(* Logix 5000 project; controller reports 1756-L63 rev 20.11; software revision 20.04; part 41 of 52 *)

        [92].log_data[45].valid := 1, [92].log_data[46].time := 3600.0, [92].log_data[46].valid := 1, [92].log_data[47].time := 3600.0, [92].log_data[47].valid := 1, [92].log_data[48].min := 6.688229, [92].log_data[48].max := 6.903953, [92].log_data[48].total := 24394.494, [92].log_data[48].time := 3600.0, [92].log_data[48].maxminute := 57, [92].log_data[48].valid := 1, [92].log_data[49].min := 7.7929306, [92].log_data[49].max := 9.600971, [92].log_data[49].total := 33255.67, [92].log_data[49].time := 3600.0, [92].log_data[49].maxminute := 51, [92].log_data[49].valid := 1, [92].log_data[50].min := 2.0512643, [92].log_data[50].max := 2.1312335, [92].log_data[50].total := 7529.347, [92].log_data[50].time := 3600.0, [92].log_data[50].minminute := 54, [92].log_data[50].valid := 1, [92].log_data[51].time := 3600.0, [92].log_data[51].valid := 1, [92].log_data[52].min := -2.9400024, [92].log_data[52].max := 0.11999512, [92].log_data[52].total := -7606.1123, [92].log_data[52].time := 3600.0, [92].log_data[52].minminute := 5, [92].log_data[52].maxminute := 4, [92].log_data[52].valid := 1, [92].log_data[53].min := -2.5, [92].log_data[53].max := 0.27999878, [92].log_data[53].total := -7261.323, [92].log_data[53].time := 3600.0, [92].log_data[53].minminute := 52, [92].log_data[53].maxminute := 30, [92].log_data[53].valid := 1, [92].log_data[54].max := 0.539, [92].log_data[54].total := 1217.2504, [92].log_data[54].time := 3600.0, [92].log_data[54].minminute := 4, [92].log_data[54].maxminute := 5, [92].log_data[54].valid := 1, [92].log_data[55].max := 0.5365, [92].log_data[55].total := 1254.4075, [92].log_data[55].time := 3600.0, [92].log_data[55].minminute := 8, [92].log_data[55].maxminute := 52, [92].log_data[55].valid := 1, [92].log_data[56].min := 0.15981378, [92].log_data[56].max := 0.16028486, [92].log_data[56].total := 576.022, [92].log_data[56].time := 3600.0, [92].log_data[56].minminute := 1, [92].log_data[56].maxminute := 14, [92].log_data[56].valid := 1, [92].log_data[57].min := 0.23891918, [92].log_data[57].max := 0.23939028,
        [92].log_data[57].total := 860.84656, [92].log_data[57].time := 3600.0, [92].log_data[57].minminute := 12, [92].log_data[57].valid := 1, [92].log_data[58].time := 3600.0, [92].log_data[58].valid := 1, [92].log_data[59].time := 3600.0, [92].log_data[59].valid := 1, [92].log_data[60].valid := 1, [92].log_data[61].valid := 1, [92].log_data[62].valid := 1, [92].log_data[63].valid := 1, [92].log_data[64].valid := 1, [92].log_data[65].valid := 1, [92].log_data[66].valid := 1, [92].log_data[67].valid := 1, [92].log_data[68].valid := 1, [92].log_data[69].valid := 1, [92].log_data[70].valid := 1, [92].log_data[71].valid := 1, [92].log_data[72].valid := 1, [92].log_data[73].valid := 1, [92].log_data[74].valid := 1, [92].log_data[75].valid := 1, [92].log_data[76].valid := 1, [92].log_data[77].valid := 1, [92].log_data[78].valid := 1, [92].log_data[79].valid := 1, [92].log_data[80].valid := 1, [92].log_data[81].valid := 1, [92].log_data[82].valid := 1, [92].log_data[83].valid := 1, [92].log_data[84].valid := 1, [92].log_data[85].valid := 1, [92].log_data[86].valid := 1, [92].log_data[87].valid := 1, [92].log_data[88].valid := 1, [92].log_data[89].valid := 1, [92].log_data[90].valid := 1, [92].log_data[91].valid := 1, [92].log_data[92].valid := 1, [92].log_data[93].valid := 1, [92].log_data[94].valid := 1, [92].log_data[95].valid := 1, [92].log_data[96].valid := 1, [92].log_data[97].valid := 1, [92].log_data[98].valid := 1, [92].log_data[99].valid := 1, [92].log_data[100].valid := 1, [92].log_data[101].valid := 1, [92].log_data[102].valid := 1, [92].log_data[103].valid := 1, [92].log_data[104].valid := 1, [92].log_data[105].valid := 1, [92].log_data[106].valid := 1, [92].log_data[107].valid := 1, [92].log_data[108].valid := 1, [92].log_data[109].valid := 1, [92].log_data[110].valid := 1, [92].log_data[111].valid := 1,
        [92].log_data[112].valid := 1, [92].log_data[113].valid := 1, [92].log_data[114].valid := 1, [92].log_data[115].valid := 1, [92].log_data[116].valid := 1, [92].log_data[117].valid := 1, [92].log_data[118].valid := 1, [92].log_data[119].valid := 1, [92].log_data[120].valid := 1, [92].log_data[121].valid := 1, [92].log_data[122].valid := 1, [92].log_data[123].valid := 1, [92].log_data[124].valid := 1, [92].time.Year := 2023, [92].time.Month := 1, [92].time.Day := 16, [92].time.Hour := 23, [92].time.Minute := 59, [92].time.Second := 59, [93].log_data[0].min := 1.0, [93].log_data[0].max := 1.0, [93].log_data[0].total := 3600.0, [93].log_data[0].time := 3600.0, [93].log_data[0].valid := 1, [93].log_data[1].max := 1.0, [93].log_data[1].total := 72.751, [93].log_data[1].time := 3600.0, [93].log_data[1].minminute := 1, [93].log_data[1].valid := 1, [93].log_data[2].max := 1.0, [93].log_data[2].total := 72.751, [93].log_data[2].time := 3600.0, [93].log_data[2].minminute := 1, [93].log_data[2].valid := 1, [93].log_data[3].time := 3600.0, [93].log_data[3].valid := 1, [93].log_data[4].time := 3600.0, [93].log_data[4].valid := 1, [93].log_data[5].max := 1.0, [93].log_data[5].total := 69.251, [93].log_data[5].time := 3600.0, [93].log_data[5].minminute := 1, [93].log_data[5].valid := 1, [93].log_data[6].time := 3600.0, [93].log_data[6].valid := 1, [93].log_data[7].time := 3600.0, [93].log_data[7].valid := 1, [93].log_data[8].min := 1.0, [93].log_data[8].max := 1.0, [93].log_data[8].total := 3600.0, [93].log_data[8].time := 3600.0, [93].log_data[8].valid := 1, [93].log_data[9].min := 1.0, [93].log_data[9].max := 1.0, [93].log_data[9].total := 3600.0, [93].log_data[9].time := 3600.0, [93].log_data[9].valid := 1, [93].log_data[10].min := 1.0, [93].log_data[10].max := 1.0, [93].log_data[10].total := 3600.0,
        [93].log_data[10].time := 3600.0, [93].log_data[10].valid := 1, [93].log_data[11].time := 3600.0, [93].log_data[11].valid := 1, [93].log_data[12].min := 1.0, [93].log_data[12].max := 1.0, [93].log_data[12].total := 3600.0, [93].log_data[12].time := 3600.0, [93].log_data[12].valid := 1, [93].log_data[13].min := 1.0, [93].log_data[13].max := 1.0, [93].log_data[13].total := 3600.0, [93].log_data[13].time := 3600.0, [93].log_data[13].valid := 1, [93].log_data[14].time := 3600.0, [93].log_data[14].valid := 1, [93].log_data[15].time := 3600.0, [93].log_data[15].valid := 1, [93].log_data[16].time := 3600.0, [93].log_data[16].valid := 1, [93].log_data[17].min := 1.0, [93].log_data[17].max := 1.0, [93].log_data[17].total := 3600.0, [93].log_data[17].time := 3600.0, [93].log_data[17].valid := 1, [93].log_data[18].time := 3600.0, [93].log_data[18].valid := 1, [93].log_data[19].time := 3600.0, [93].log_data[19].valid := 1, [93].log_data[20].time := 3600.0, [93].log_data[20].valid := 1, [93].log_data[21].min := 1.0, [93].log_data[21].max := 1.0, [93].log_data[21].total := 3600.0, [93].log_data[21].time := 3600.0, [93].log_data[21].valid := 1, [93].log_data[22].time := 3600.0, [93].log_data[22].valid := 1, [93].log_data[23].time := 3600.0, [93].log_data[23].valid := 1, [93].log_data[24].time := 3600.0, [93].log_data[24].valid := 1, [93].log_data[25].time := 3600.0, [93].log_data[25].valid := 1, [93].log_data[26].time := 3600.0, [93].log_data[26].valid := 1, [93].log_data[27].time := 3600.0, [93].log_data[27].valid := 1, [93].log_data[28].time := 3600.0, [93].log_data[28].valid := 1, [93].log_data[29].min := 1.0, [93].log_data[29].max := 1.0, [93].log_data[29].total := 3600.0, [93].log_data[29].time := 3600.0, [93].log_data[29].valid := 1, [93].log_data[30].min := 1.0, [93].log_data[30].max := 1.0, [93].log_data[30].total := 3600.0, [93].log_data[30].time := 3600.0, [93].log_data[30].valid := 1,
        [93].log_data[31].max := 1.0, [93].log_data[31].total := 1629.7471, [93].log_data[31].time := 3600.0, [93].log_data[31].maxminute := 8, [93].log_data[31].valid := 1, [93].log_data[32].max := 1.0, [93].log_data[32].total := 1529.249, [93].log_data[32].time := 3600.0, [93].log_data[32].minminute := 7, [93].log_data[32].valid := 1, [93].log_data[33].time := 3600.0, [93].log_data[33].valid := 1, [93].log_data[34].time := 3600.0, [93].log_data[34].valid := 1, [93].log_data[35].max := 1.0, [93].log_data[35].total := 1440.498, [93].log_data[35].time := 3600.0, [93].log_data[35].minminute := 1, [93].log_data[35].valid := 1, [93].log_data[36].max := 1.0, [93].log_data[36].total := 1629.7471, [93].log_data[36].time := 3600.0, [93].log_data[36].maxminute := 2, [93].log_data[36].valid := 1, [93].log_data[37].max := 7.1119633, [93].log_data[37].total := 82.35939, [93].log_data[37].time := 3600.0, [93].log_data[37].valid := 1, [93].log_data[38].time := 3600.0, [93].log_data[38].valid := 1, [93].log_data[39].min := 0.99494183, [93].log_data[39].max := 1.0174367, [93].log_data[39].total := 3603.3508, [93].log_data[39].time := 3600.0, [93].log_data[39].minminute := 5, [93].log_data[39].valid := 1, [93].log_data[40].min := 7.5802555, [93].log_data[40].max := 7.604989, [93].log_data[40].total := 27354.303, [93].log_data[40].time := 3600.0, [93].log_data[40].minminute := 6, [93].log_data[40].maxminute := 8, [93].log_data[40].valid := 1, [93].log_data[41].min := 0.022540038, [93].log_data[41].max := 0.026073486, [93].log_data[41].total := 83.22505, [93].log_data[41].time := 3600.0, [93].log_data[41].minminute := 43, [93].log_data[41].maxminute := 56, [93].log_data[41].valid := 1, [93].log_data[42].min := 2.2917604, [93].log_data[42].max := 2.296236, [93].log_data[42].total := 8259.312, [93].log_data[42].time := 3600.0, [93].log_data[42].minminute := 4, [93].log_data[42].maxminute := 33, [93].log_data[42].valid := 1, [93].log_data[43].min := -0.27999878, [93].log_data[43].max := -0.26000214, [93].log_data[43].total := -1001.4477,
        [93].log_data[43].time := 3600.0, [93].log_data[43].valid := 1, [93].log_data[44].min := -0.3199997, [93].log_data[44].max := -0.30000305, [93].log_data[44].total := -1080.1111, [93].log_data[44].time := 3600.0, [93].log_data[44].minminute := 37, [93].log_data[44].valid := 1, [93].log_data[45].time := 3600.0, [93].log_data[45].valid := 1, [93].log_data[46].time := 3600.0, [93].log_data[46].valid := 1, [93].log_data[47].time := 3600.0, [93].log_data[47].valid := 1, [93].log_data[48].min := 6.587924, [93].log_data[48].max := 6.9380293, [93].log_data[48].total := 24235.338, [93].log_data[48].time := 3600.0, [93].log_data[48].minminute := 26, [93].log_data[48].maxminute := 1, [93].log_data[48].valid := 1, [93].log_data[49].min := 6.965759, [93].log_data[49].max := 9.442367, [93].log_data[49].total := 29303.482, [93].log_data[49].time := 3600.0, [93].log_data[49].minminute := 22, [93].log_data[49].maxminute := 59, [93].log_data[49].valid := 1, [93].log_data[50].min := 2.0797658, [93].log_data[50].max := 2.1550238, [93].log_data[50].total := 7630.34, [93].log_data[50].time := 3600.0, [93].log_data[50].minminute := 59, [93].log_data[50].maxminute := 3, [93].log_data[50].valid := 1, [93].log_data[51].time := 3600.0, [93].log_data[51].valid := 1, [93].log_data[52].min := -3.1200027, [93].log_data[52].max := 0.11999512, [93].log_data[52].total := -7898.7217, [93].log_data[52].time := 3600.0, [93].log_data[52].minminute := 29, [93].log_data[52].maxminute := 7, [93].log_data[52].valid := 1, [93].log_data[53].min := -2.5200043, [93].log_data[53].max := 0.27999878, [93].log_data[53].total := -7128.1104, [93].log_data[53].time := 3600.0, [93].log_data[53].minminute := 13, [93].log_data[53].maxminute := 23, [93].log_data[53].valid := 1, [93].log_data[54].max := 0.5565, [93].log_data[54].total := 1254.5945, [93].log_data[54].time := 3600.0, [93].log_data[54].minminute := 7, [93].log_data[54].maxminute := 30, [93].log_data[54].valid := 1, [93].log_data[55].max := 0.519, [93].log_data[55].total := 1216.6926, [93].log_data[55].time := 3600.0,
        [93].log_data[55].minminute := 1, [93].log_data[55].maxminute := 44, [93].log_data[55].valid := 1, [93].log_data[56].min := 0.15981378, [93].log_data[56].max := 0.16024561, [93].log_data[56].total := 575.9473, [93].log_data[56].time := 3600.0, [93].log_data[56].minminute := 24, [93].log_data[56].maxminute := 41, [93].log_data[56].valid := 1, [93].log_data[57].min := 0.23754516, [93].log_data[57].max := 0.23935102, [93].log_data[57].total := 858.23517, [93].log_data[57].time := 3600.0, [93].log_data[57].minminute := 39, [93].log_data[57].maxminute := 21, [93].log_data[57].valid := 1, [93].log_data[58].time := 3600.0, [93].log_data[58].valid := 1, [93].log_data[59].time := 3600.0, [93].log_data[59].valid := 1, [93].log_data[60].valid := 1, [93].log_data[61].valid := 1, [93].log_data[62].valid := 1, [93].log_data[63].valid := 1, [93].log_data[64].valid := 1, [93].log_data[65].valid := 1, [93].log_data[66].valid := 1, [93].log_data[67].valid := 1, [93].log_data[68].valid := 1, [93].log_data[69].valid := 1, [93].log_data[70].valid := 1, [93].log_data[71].valid := 1, [93].log_data[72].valid := 1, [93].log_data[73].valid := 1, [93].log_data[74].valid := 1, [93].log_data[75].valid := 1, [93].log_data[76].valid := 1, [93].log_data[77].valid := 1, [93].log_data[78].valid := 1, [93].log_data[79].valid := 1, [93].log_data[80].valid := 1, [93].log_data[81].valid := 1, [93].log_data[82].valid := 1, [93].log_data[83].valid := 1, [93].log_data[84].valid := 1, [93].log_data[85].valid := 1, [93].log_data[86].valid := 1, [93].log_data[87].valid := 1, [93].log_data[88].valid := 1, [93].log_data[89].valid := 1, [93].log_data[90].valid := 1, [93].log_data[91].valid := 1, [93].log_data[92].valid := 1, [93].log_data[93].valid := 1, [93].log_data[94].valid := 1, [93].log_data[95].valid := 1, [93].log_data[96].valid := 1, [93].log_data[97].valid := 1, [93].log_data[98].valid := 1,
        [93].log_data[99].valid := 1, [93].log_data[100].valid := 1, [93].log_data[101].valid := 1, [93].log_data[102].valid := 1, [93].log_data[103].valid := 1, [93].log_data[104].valid := 1, [93].log_data[105].valid := 1, [93].log_data[106].valid := 1, [93].log_data[107].valid := 1, [93].log_data[108].valid := 1, [93].log_data[109].valid := 1, [93].log_data[110].valid := 1, [93].log_data[111].valid := 1, [93].log_data[112].valid := 1, [93].log_data[113].valid := 1, [93].log_data[114].valid := 1, [93].log_data[115].valid := 1, [93].log_data[116].valid := 1, [93].log_data[117].valid := 1, [93].log_data[118].valid := 1, [93].log_data[119].valid := 1, [93].log_data[120].valid := 1, [93].log_data[121].valid := 1, [93].log_data[122].valid := 1, [93].log_data[123].valid := 1, [93].log_data[124].valid := 1, [93].time.Year := 2023, [93].time.Month := 1, [93].time.Day := 17, [93].time.Minute := 59, [93].time.Second := 59, [94].log_data[0].min := 1.0, [94].log_data[0].max := 1.0, [94].log_data[0].total := 3600.0, [94].log_data[0].time := 3600.0, [94].log_data[0].valid := 1, [94].log_data[1].time := 3600.0, [94].log_data[1].valid := 1, [94].log_data[2].time := 3600.0, [94].log_data[2].valid := 1, [94].log_data[3].time := 3600.0, [94].log_data[3].valid := 1, [94].log_data[4].time := 3600.0, [94].log_data[4].valid := 1, [94].log_data[5].time := 3600.0, [94].log_data[5].valid := 1, [94].log_data[6].time := 3600.0, [94].log_data[6].valid := 1, [94].log_data[7].time := 3600.0, [94].log_data[7].valid := 1, [94].log_data[8].max := 1.0, [94].log_data[8].total := 2725.751, [94].log_data[8].time := 3600.0, [94].log_data[8].minminute := 45, [94].log_data[8].valid := 1, [94].log_data[9].max := 1.0, [94].log_data[9].total := 2725.751, [94].log_data[9].time := 3600.0, [94].log_data[9].minminute := 45, [94].log_data[9].valid := 1,
        [94].log_data[10].min := 1.0, [94].log_data[10].max := 1.0, [94].log_data[10].total := 3600.0, [94].log_data[10].time := 3600.0, [94].log_data[10].valid := 1, [94].log_data[11].time := 3600.0, [94].log_data[11].valid := 1, [94].log_data[12].min := 1.0, [94].log_data[12].max := 1.0, [94].log_data[12].total := 3600.0, [94].log_data[12].time := 3600.0, [94].log_data[12].valid := 1, [94].log_data[13].min := 1.0, [94].log_data[13].max := 1.0, [94].log_data[13].total := 3600.0, [94].log_data[13].time := 3600.0, [94].log_data[13].valid := 1, [94].log_data[14].time := 3600.0, [94].log_data[14].valid := 1, [94].log_data[15].time := 3600.0, [94].log_data[15].valid := 1, [94].log_data[16].time := 3600.0, [94].log_data[16].valid := 1, [94].log_data[17].min := 1.0, [94].log_data[17].max := 1.0, [94].log_data[17].total := 3600.0, [94].log_data[17].time := 3600.0, [94].log_data[17].valid := 1, [94].log_data[18].time := 3600.0, [94].log_data[18].valid := 1, [94].log_data[19].time := 3600.0, [94].log_data[19].valid := 1, [94].log_data[20].time := 3600.0, [94].log_data[20].valid := 1, [94].log_data[21].min := 1.0, [94].log_data[21].max := 1.0, [94].log_data[21].total := 3600.0, [94].log_data[21].time := 3600.0, [94].log_data[21].valid := 1, [94].log_data[22].time := 3600.0, [94].log_data[22].valid := 1, [94].log_data[23].time := 3600.0, [94].log_data[23].valid := 1, [94].log_data[24].time := 3600.0, [94].log_data[24].valid := 1, [94].log_data[25].time := 3600.0, [94].log_data[25].valid := 1, [94].log_data[26].time := 3600.0, [94].log_data[26].valid := 1, [94].log_data[27].time := 3600.0, [94].log_data[27].valid := 1, [94].log_data[28].time := 3600.0, [94].log_data[28].valid := 1, [94].log_data[29].min := 1.0, [94].log_data[29].max := 1.0, [94].log_data[29].total := 3600.0, [94].log_data[29].time := 3600.0, [94].log_data[29].valid := 1, [94].log_data[30].min := 1.0, [94].log_data[30].max := 1.0,
        [94].log_data[30].total := 3600.0, [94].log_data[30].time := 3600.0, [94].log_data[30].valid := 1, [94].log_data[31].max := 1.0, [94].log_data[31].total := 1086.498, [94].log_data[31].time := 3600.0, [94].log_data[31].maxminute := 11, [94].log_data[31].valid := 1, [94].log_data[32].max := 1.0, [94].log_data[32].total := 1201.7471, [94].log_data[32].time := 3600.0, [94].log_data[32].maxminute := 1, [94].log_data[32].valid := 1, [94].log_data[33].time := 3600.0, [94].log_data[33].valid := 1, [94].log_data[34].time := 3600.0, [94].log_data[34].valid := 1, [94].log_data[35].max := 1.0, [94].log_data[35].total := 1289.998, [94].log_data[35].time := 3600.0, [94].log_data[35].minminute := 4, [94].log_data[35].valid := 1, [94].log_data[36].max := 1.0, [94].log_data[36].total := 1086.498, [94].log_data[36].time := 3600.0, [94].log_data[36].maxminute := 5, [94].log_data[36].valid := 1, [94].log_data[37].time := 3600.0, [94].log_data[37].valid := 1, [94].log_data[38].time := 3600.0, [94].log_data[38].valid := 1, [94].log_data[39].min := 0.9944707, [94].log_data[39].max := 1.0054238, [94].log_data[39].total := 3603.0454, [94].log_data[39].time := 3600.0, [94].log_data[39].minminute := 12, [94].log_data[39].valid := 1, [94].log_data[40].min := 7.591522, [94].log_data[40].max := 7.604989, [94].log_data[40].total := 27355.736, [94].log_data[40].time := 3600.0, [94].log_data[40].minminute := 48, [94].log_data[40].maxminute := 54, [94].log_data[40].valid := 1, [94].log_data[41].min := 0.02273633, [94].log_data[41].max := 0.026073486, [94].log_data[41].total := 83.72127, [94].log_data[41].time := 3600.0, [94].log_data[41].minminute := 9, [94].log_data[41].valid := 1, [94].log_data[42].min := 2.2911716, [94].log_data[42].max := 2.2963536, [94].log_data[42].total := 8259.223, [94].log_data[42].time := 3600.0, [94].log_data[42].minminute := 33, [94].log_data[42].maxminute := 35, [94].log_data[42].valid := 1, [94].log_data[43].min := -0.27999878, [94].log_data[43].max := -0.26000214, [94].log_data[43].total := -1002.2216,
        [94].log_data[43].time := 3600.0, [94].log_data[43].valid := 1, [94].log_data[44].min := -0.3199997, [94].log_data[44].max := -0.30000305, [94].log_data[44].total := -1080.0962, [94].log_data[44].time := 3600.0, [94].log_data[44].minminute := 20, [94].log_data[44].valid := 1, [94].log_data[45].time := 3600.0, [94].log_data[45].valid := 1, [94].log_data[46].time := 3600.0, [94].log_data[46].valid := 1, [94].log_data[47].time := 3600.0, [94].log_data[47].valid := 1, [94].log_data[48].min := 6.7649, [94].log_data[48].max := 6.7800145, [94].log_data[48].total := 24376.885, [94].log_data[48].time := 3600.0, [94].log_data[48].minminute := 50, [94].log_data[48].maxminute := 1, [94].log_data[48].valid := 1, [94].log_data[49].min := 9.429412, [94].log_data[49].max := 9.602148, [94].log_data[49].total := 34382.223, [94].log_data[49].time := 3600.0, [94].log_data[49].maxminute := 32, [94].log_data[49].valid := 1, [94].log_data[50].min := 1.9999144, [94].log_data[50].max := 2.1160402, [94].log_data[50].total := 7404.776, [94].log_data[50].time := 3600.0, [94].log_data[50].minminute := 45, [94].log_data[50].maxminute := 59, [94].log_data[50].valid := 1, [94].log_data[51].time := 3600.0, [94].log_data[51].valid := 1, [94].log_data[52].min := -2.9400024, [94].log_data[52].max := 0.11999512, [94].log_data[52].total := -6819.65, [94].log_data[52].time := 3600.0, [94].log_data[52].minminute := 12, [94].log_data[52].valid := 1, [94].log_data[53].min := -2.4800034, [94].log_data[53].max := 0.27999878, [94].log_data[53].total := -6552.212, [94].log_data[53].time := 3600.0, [94].log_data[53].minminute := 2, [94].log_data[53].maxminute := 5, [94].log_data[53].valid := 1, [94].log_data[54].max := 0.524, [94].log_data[54].total := 906.4553, [94].log_data[54].time := 3600.0, [94].log_data[54].maxminute := 12, [94].log_data[54].valid := 1, [94].log_data[55].max := 0.517, [94].log_data[55].total := 943.5342, [94].log_data[55].time := 3600.0, [94].log_data[55].minminute := 4, [94].log_data[55].maxminute := 5, [94].log_data[55].valid := 1,
        [94].log_data[56].min := 0.15985303, [94].log_data[56].max := 0.16024561, [94].log_data[56].total := 575.978, [94].log_data[56].time := 3600.0, [94].log_data[56].minminute := 5, [94].log_data[56].maxminute := 25, [94].log_data[56].valid := 1, [94].log_data[57].min := 0.23754516, [94].log_data[57].max := 0.237977, [94].log_data[57].total := 855.8624, [94].log_data[57].time := 3600.0, [94].log_data[57].minminute := 21, [94].log_data[57].maxminute := 44, [94].log_data[57].valid := 1, [94].log_data[58].time := 3600.0, [94].log_data[58].valid := 1, [94].log_data[59].time := 3600.0, [94].log_data[59].valid := 1, [94].log_data[60].valid := 1, [94].log_data[61].valid := 1, [94].log_data[62].valid := 1, [94].log_data[63].valid := 1, [94].log_data[64].valid := 1, [94].log_data[65].valid := 1, [94].log_data[66].valid := 1, [94].log_data[67].valid := 1, [94].log_data[68].valid := 1, [94].log_data[69].valid := 1, [94].log_data[70].valid := 1, [94].log_data[71].valid := 1, [94].log_data[72].valid := 1, [94].log_data[73].valid := 1, [94].log_data[74].valid := 1, [94].log_data[75].valid := 1, [94].log_data[76].valid := 1, [94].log_data[77].valid := 1, [94].log_data[78].valid := 1, [94].log_data[79].valid := 1, [94].log_data[80].valid := 1, [94].log_data[81].valid := 1, [94].log_data[82].valid := 1, [94].log_data[83].valid := 1, [94].log_data[84].valid := 1, [94].log_data[85].valid := 1, [94].log_data[86].valid := 1, [94].log_data[87].valid := 1, [94].log_data[88].valid := 1, [94].log_data[89].valid := 1, [94].log_data[90].valid := 1, [94].log_data[91].valid := 1, [94].log_data[92].valid := 1, [94].log_data[93].valid := 1, [94].log_data[94].valid := 1, [94].log_data[95].valid := 1, [94].log_data[96].valid := 1, [94].log_data[97].valid := 1, [94].log_data[98].valid := 1, [94].log_data[99].valid := 1, [94].log_data[100].valid := 1, [94].log_data[101].valid := 1,
        [94].log_data[102].valid := 1, [94].log_data[103].valid := 1, [94].log_data[104].valid := 1, [94].log_data[105].valid := 1, [94].log_data[106].valid := 1, [94].log_data[107].valid := 1, [94].log_data[108].valid := 1, [94].log_data[109].valid := 1, [94].log_data[110].valid := 1, [94].log_data[111].valid := 1, [94].log_data[112].valid := 1, [94].log_data[113].valid := 1, [94].log_data[114].valid := 1, [94].log_data[115].valid := 1, [94].log_data[116].valid := 1, [94].log_data[117].valid := 1, [94].log_data[118].valid := 1, [94].log_data[119].valid := 1, [94].log_data[120].valid := 1, [94].log_data[121].valid := 1, [94].log_data[122].valid := 1, [94].log_data[123].valid := 1, [94].log_data[124].valid := 1, [94].time.Year := 2023, [94].time.Month := 1, [94].time.Day := 17, [94].time.Hour := 1, [94].time.Minute := 59, [94].time.Second := 59, [95].log_data[0].min := 1.0, [95].log_data[0].max := 1.0, [95].log_data[0].total := 3600.0, [95].log_data[0].time := 3600.0, [95].log_data[0].valid := 1, [95].log_data[1].max := 1.0, [95].log_data[1].total := 526.5, [95].log_data[1].time := 3600.0, [95].log_data[1].maxminute := 3, [95].log_data[1].valid := 1, [95].log_data[2].max := 1.0, [95].log_data[2].total := 523.0, [95].log_data[2].time := 3600.0, [95].log_data[2].maxminute := 3, [95].log_data[2].valid := 1, [95].log_data[3].time := 3600.0, [95].log_data[3].valid := 1, [95].log_data[4].time := 3600.0, [95].log_data[4].valid := 1, [95].log_data[5].max := 1.0, [95].log_data[5].total := 233.0, [95].log_data[5].time := 3600.0, [95].log_data[5].maxminute := 5, [95].log_data[5].valid := 1, [95].log_data[6].time := 3600.0, [95].log_data[6].valid := 1, [95].log_data[7].time := 3600.0, [95].log_data[7].valid := 1, [95].log_data[8].max := 1.0, [95].log_data[8].total := 3184.749, [95].log_data[8].time := 3600.0,
        [95].log_data[8].maxminute := 6, [95].log_data[8].valid := 1, [95].log_data[9].max := 1.0, [95].log_data[9].total := 3181.249, [95].log_data[9].time := 3600.0, [95].log_data[9].maxminute := 6, [95].log_data[9].valid := 1, [95].log_data[10].min := 1.0, [95].log_data[10].max := 1.0, [95].log_data[10].total := 3600.0, [95].log_data[10].time := 3600.0, [95].log_data[10].valid := 1, [95].log_data[11].time := 3600.0, [95].log_data[11].valid := 1, [95].log_data[12].min := 1.0, [95].log_data[12].max := 1.0, [95].log_data[12].total := 3600.0, [95].log_data[12].time := 3600.0, [95].log_data[12].valid := 1, [95].log_data[13].min := 1.0, [95].log_data[13].max := 1.0, [95].log_data[13].total := 3600.0, [95].log_data[13].time := 3600.0, [95].log_data[13].valid := 1, [95].log_data[14].time := 3600.0, [95].log_data[14].valid := 1, [95].log_data[15].time := 3600.0, [95].log_data[15].valid := 1, [95].log_data[16].time := 3600.0, [95].log_data[16].valid := 1, [95].log_data[17].min := 1.0, [95].log_data[17].max := 1.0, [95].log_data[17].total := 3600.0, [95].log_data[17].time := 3600.0, [95].log_data[17].valid := 1, [95].log_data[18].time := 3600.0, [95].log_data[18].valid := 1, [95].log_data[19].time := 3600.0, [95].log_data[19].valid := 1, [95].log_data[20].time := 3600.0, [95].log_data[20].valid := 1, [95].log_data[21].min := 1.0, [95].log_data[21].max := 1.0, [95].log_data[21].total := 3600.0, [95].log_data[21].time := 3600.0, [95].log_data[21].valid := 1, [95].log_data[22].time := 3600.0, [95].log_data[22].valid := 1, [95].log_data[23].time := 3600.0, [95].log_data[23].valid := 1, [95].log_data[24].time := 3600.0, [95].log_data[24].valid := 1, [95].log_data[25].time := 3600.0, [95].log_data[25].valid := 1, [95].log_data[26].time := 3600.0, [95].log_data[26].valid := 1, [95].log_data[27].time := 3600.0, [95].log_data[27].valid := 1, [95].log_data[28].time := 3600.0, [95].log_data[28].valid := 1,
        [95].log_data[29].min := 1.0, [95].log_data[29].max := 1.0, [95].log_data[29].total := 3600.0, [95].log_data[29].time := 3600.0, [95].log_data[29].valid := 1, [95].log_data[30].min := 1.0, [95].log_data[30].max := 1.0, [95].log_data[30].total := 3600.0, [95].log_data[30].time := 3600.0, [95].log_data[30].valid := 1, [95].log_data[31].max := 1.0, [95].log_data[31].total := 1514.247, [95].log_data[31].time := 3600.0, [95].log_data[31].maxminute := 7, [95].log_data[31].valid := 1, [95].log_data[32].max := 1.0, [95].log_data[32].total := 1221.998, [95].log_data[32].time := 3600.0, [95].log_data[32].maxminute := 15, [95].log_data[32].valid := 1, [95].log_data[33].time := 3600.0, [95].log_data[33].valid := 1, [95].log_data[34].time := 3600.0, [95].log_data[34].valid := 1, [95].log_data[35].max := 1.0, [95].log_data[35].total := 1593.7471, [95].log_data[35].time := 3600.0, [95].log_data[35].maxminute := 9, [95].log_data[35].valid := 1, [95].log_data[36].max := 1.0, [95].log_data[36].total := 1139.247, [95].log_data[36].time := 3600.0, [95].log_data[36].maxminute := 7, [95].log_data[36].valid := 1, [95].log_data[37].max := 7.4978714, [95].log_data[37].total := 3407.6616, [95].log_data[37].time := 3600.0, [95].log_data[37].maxminute := 4, [95].log_data[37].valid := 1, [95].log_data[38].time := 3600.0, [95].log_data[38].valid := 1, [95].log_data[39].min := 0.99282193, [95].log_data[39].max := 1.0216767, [95].log_data[39].total := 3605.1196, [95].log_data[39].time := 3600.0, [95].log_data[39].minminute := 54, [95].log_data[39].maxminute := 10, [95].log_data[39].valid := 1, [95].log_data[40].min := 7.591522, [95].log_data[40].max := 7.605263, [95].log_data[40].total := 27359.295, [95].log_data[40].time := 3600.0, [95].log_data[40].minminute := 6, [95].log_data[40].maxminute := 11, [95].log_data[40].valid := 1, [95].log_data[41].min := 0.022540038, [95].log_data[41].max := 0.027054932, [95].log_data[41].total := 83.72717, [95].log_data[41].time := 3600.0, [95].log_data[41].minminute := 19,
        [95].log_data[41].maxminute := 36, [95].log_data[41].valid := 1, [95].log_data[42].min := 2.291525, [95].log_data[42].max := 2.296118, [95].log_data[42].total := 8259.106, [95].log_data[42].time := 3600.0, [95].log_data[42].minminute := 11, [95].log_data[42].maxminute := 11, [95].log_data[42].valid := 1, [95].log_data[43].min := -0.27999878, [95].log_data[43].max := -0.26000214, [95].log_data[43].total := -976.2031, [95].log_data[43].time := 3600.0, [95].log_data[43].valid := 1, [95].log_data[44].min := -0.30000305, [95].log_data[44].max := -0.30000305, [95].log_data[44].total := -1080.0911, [95].log_data[44].time := 3600.0, [95].log_data[44].valid := 1, [95].log_data[45].time := 3600.0, [95].log_data[45].valid := 1, [95].log_data[46].time := 3600.0, [95].log_data[46].valid := 1, [95].log_data[47].time := 3600.0, [95].log_data[47].valid := 1, [95].log_data[48].min := 6.589573, [95].log_data[48].max := 6.9465485, [95].log_data[48].total := 24249.084, [95].log_data[48].time := 3600.0, [95].log_data[48].minminute := 37, [95].log_data[48].maxminute := 12, [95].log_data[48].valid := 1, [95].log_data[49].min := 6.8835125, [95].log_data[49].max := 9.557198, [95].log_data[49].total := 29212.176, [95].log_data[49].time := 3600.0, [95].log_data[49].minminute := 32, [95].log_data[49].maxminute := 2, [95].log_data[49].valid := 1, [95].log_data[50].min := 2.0484376, [95].log_data[50].max := 2.150313, [95].log_data[50].total := 7525.7383, [95].log_data[50].time := 3600.0, [95].log_data[50].minminute := 59, [95].log_data[50].maxminute := 6, [95].log_data[50].valid := 1, [95].log_data[51].time := 3600.0, [95].log_data[51].valid := 1, [95].log_data[52].min := -4.3399963, [95].log_data[52].max := 0.11999512, [95].log_data[52].total := -7494.401, [95].log_data[52].time := 3600.0, [95].log_data[52].minminute := 7, [95].log_data[52].maxminute := 14, [95].log_data[52].valid := 1, [95].log_data[53].min := -3.9399948, [95].log_data[53].max := 0.27999878, [95].log_data[53].total := -6960.026, [95].log_data[53].time := 3600.0, [95].log_data[53].minminute := 7,
        [95].log_data[53].maxminute := 19, [95].log_data[53].valid := 1, [95].log_data[54].max := 0.5355, [95].log_data[54].total := 1083.5779, [95].log_data[54].time := 3600.0, [95].log_data[54].maxminute := 26, [95].log_data[54].valid := 1, [95].log_data[55].max := 0.518, [95].log_data[55].total := 1081.9321, [95].log_data[55].time := 3600.0, [95].log_data[55].maxminute := 30, [95].log_data[55].valid := 1, [95].log_data[56].min := 0.15973525, [95].log_data[56].max := 0.16020635, [95].log_data[56].total := 575.83905, [95].log_data[56].time := 3600.0, [95].log_data[56].minminute := 37, [95].log_data[56].maxminute := 4, [95].log_data[56].valid := 1, [95].log_data[57].min := 0.2362104, [95].log_data[57].max := 0.23801626, [95].log_data[57].total := 854.2079, [95].log_data[57].time := 3600.0, [95].log_data[57].minminute := 52, [95].log_data[57].maxminute := 15, [95].log_data[57].valid := 1, [95].log_data[58].time := 3600.0, [95].log_data[58].valid := 1, [95].log_data[59].time := 3600.0, [95].log_data[59].valid := 1, [95].log_data[60].valid := 1, [95].log_data[61].valid := 1, [95].log_data[62].valid := 1, [95].log_data[63].valid := 1, [95].log_data[64].valid := 1, [95].log_data[65].valid := 1, [95].log_data[66].valid := 1, [95].log_data[67].valid := 1, [95].log_data[68].valid := 1, [95].log_data[69].valid := 1, [95].log_data[70].valid := 1, [95].log_data[71].valid := 1, [95].log_data[72].valid := 1, [95].log_data[73].valid := 1, [95].log_data[74].valid := 1, [95].log_data[75].valid := 1, [95].log_data[76].valid := 1, [95].log_data[77].valid := 1, [95].log_data[78].valid := 1, [95].log_data[79].valid := 1, [95].log_data[80].valid := 1, [95].log_data[81].valid := 1, [95].log_data[82].valid := 1, [95].log_data[83].valid := 1, [95].log_data[84].valid := 1, [95].log_data[85].valid := 1, [95].log_data[86].valid := 1, [95].log_data[87].valid := 1, [95].log_data[88].valid := 1, [95].log_data[89].valid := 1,
        [95].log_data[90].valid := 1, [95].log_data[91].valid := 1, [95].log_data[92].valid := 1, [95].log_data[93].valid := 1, [95].log_data[94].valid := 1, [95].log_data[95].valid := 1, [95].log_data[96].valid := 1, [95].log_data[97].valid := 1, [95].log_data[98].valid := 1, [95].log_data[99].valid := 1, [95].log_data[100].valid := 1, [95].log_data[101].valid := 1, [95].log_data[102].valid := 1, [95].log_data[103].valid := 1, [95].log_data[104].valid := 1, [95].log_data[105].valid := 1, [95].log_data[106].valid := 1, [95].log_data[107].valid := 1, [95].log_data[108].valid := 1, [95].log_data[109].valid := 1, [95].log_data[110].valid := 1, [95].log_data[111].valid := 1, [95].log_data[112].valid := 1, [95].log_data[113].valid := 1, [95].log_data[114].valid := 1, [95].log_data[115].valid := 1, [95].log_data[116].valid := 1, [95].log_data[117].valid := 1, [95].log_data[118].valid := 1, [95].log_data[119].valid := 1, [95].log_data[120].valid := 1, [95].log_data[121].valid := 1, [95].log_data[122].valid := 1, [95].log_data[123].valid := 1, [95].log_data[124].valid := 1, [95].time.Year := 2023, [95].time.Month := 1, [95].time.Day := 17, [95].time.Hour := 2, [95].time.Minute := 59, [95].time.Second := 59, [96].log_data[0].min := 1.0, [96].log_data[0].max := 1.0, [96].log_data[0].total := 3600.0, [96].log_data[0].time := 3600.0, [96].log_data[0].valid := 1, [96].log_data[1].time := 3600.0, [96].log_data[1].valid := 1, [96].log_data[2].time := 3600.0, [96].log_data[2].valid := 1, [96].log_data[3].time := 3600.0, [96].log_data[3].valid := 1, [96].log_data[4].time := 3600.0, [96].log_data[4].valid := 1, [96].log_data[5].time := 3600.0, [96].log_data[5].valid := 1, [96].log_data[6].time := 3600.0, [96].log_data[6].valid := 1, [96].log_data[7].time := 3600.0, [96].log_data[7].valid := 1,
        [96].log_data[8].max := 1.0, [96].log_data[8].total := 2187.751, [96].log_data[8].time := 3600.0, [96].log_data[8].minminute := 36, [96].log_data[8].valid := 1, [96].log_data[9].max := 1.0, [96].log_data[9].total := 2187.751, [96].log_data[9].time := 3600.0, [96].log_data[9].minminute := 36, [96].log_data[9].valid := 1, [96].log_data[10].min := 1.0, [96].log_data[10].max := 1.0, [96].log_data[10].total := 3600.0, [96].log_data[10].time := 3600.0, [96].log_data[10].valid := 1, [96].log_data[11].time := 3600.0, [96].log_data[11].valid := 1, [96].log_data[12].min := 1.0, [96].log_data[12].max := 1.0, [96].log_data[12].total := 3600.0, [96].log_data[12].time := 3600.0, [96].log_data[12].valid := 1, [96].log_data[13].min := 1.0, [96].log_data[13].max := 1.0, [96].log_data[13].total := 3600.0, [96].log_data[13].time := 3600.0, [96].log_data[13].valid := 1, [96].log_data[14].time := 3600.0, [96].log_data[14].valid := 1, [96].log_data[15].time := 3600.0, [96].log_data[15].valid := 1, [96].log_data[16].time := 3600.0, [96].log_data[16].valid := 1, [96].log_data[17].min := 1.0, [96].log_data[17].max := 1.0, [96].log_data[17].total := 3600.0, [96].log_data[17].time := 3600.0, [96].log_data[17].valid := 1, [96].log_data[18].time := 3600.0, [96].log_data[18].valid := 1, [96].log_data[19].time := 3600.0, [96].log_data[19].valid := 1, [96].log_data[20].time := 3600.0, [96].log_data[20].valid := 1, [96].log_data[21].min := 1.0, [96].log_data[21].max := 1.0, [96].log_data[21].total := 3600.0, [96].log_data[21].time := 3600.0, [96].log_data[21].valid := 1, [96].log_data[22].time := 3600.0, [96].log_data[22].valid := 1, [96].log_data[23].time := 3600.0, [96].log_data[23].valid := 1, [96].log_data[24].time := 3600.0, [96].log_data[24].valid := 1, [96].log_data[25].time := 3600.0, [96].log_data[25].valid := 1, [96].log_data[26].time := 3600.0, [96].log_data[26].valid := 1, [96].log_data[27].time := 3600.0,
        [96].log_data[27].valid := 1, [96].log_data[28].time := 3600.0, [96].log_data[28].valid := 1, [96].log_data[29].min := 1.0, [96].log_data[29].max := 1.0, [96].log_data[29].total := 3600.0, [96].log_data[29].time := 3600.0, [96].log_data[29].valid := 1, [96].log_data[30].min := 1.0, [96].log_data[30].max := 1.0, [96].log_data[30].total := 3600.0, [96].log_data[30].time := 3600.0, [96].log_data[30].valid := 1, [96].log_data[31].max := 1.0, [96].log_data[31].total := 975.49805, [96].log_data[31].time := 3600.0, [96].log_data[31].maxminute := 8, [96].log_data[31].valid := 1, [96].log_data[32].max := 1.0, [96].log_data[32].total := 951.5, [96].log_data[32].time := 3600.0, [96].log_data[32].minminute := 6, [96].log_data[32].valid := 1, [96].log_data[33].time := 3600.0, [96].log_data[33].valid := 1, [96].log_data[34].time := 3600.0, [96].log_data[34].valid := 1, [96].log_data[35].max := 1.0, [96].log_data[35].total := 751.99805, [96].log_data[35].time := 3600.0, [96].log_data[35].valid := 1, [96].log_data[36].max := 1.0, [96].log_data[36].total := 1086.498, [96].log_data[36].time := 3600.0, [96].log_data[36].maxminute := 2, [96].log_data[36].valid := 1, [96].log_data[37].time := 3600.0, [96].log_data[37].valid := 1, [96].log_data[38].time := 3600.0, [96].log_data[38].valid := 1, [96].log_data[39].min := 0.9938818, [96].log_data[39].max := 1.0050704, [96].log_data[39].total := 3599.581, [96].log_data[39].time := 3600.0, [96].log_data[39].minminute := 26, [96].log_data[39].maxminute := 50, [96].log_data[39].valid := 1, [96].log_data[40].min := 7.591522, [96].log_data[40].max := 7.603339, [96].log_data[40].total := 27357.35, [96].log_data[40].time := 3600.0, [96].log_data[40].minminute := 52, [96].log_data[40].maxminute := 57, [96].log_data[40].valid := 1, [96].log_data[41].min := 0.02273633, [96].log_data[41].max := 0.025091797, [96].log_data[41].total := 83.03872, [96].log_data[41].time := 3600.0, [96].log_data[41].maxminute := 4, [96].log_data[41].valid := 1,
        [96].log_data[42].min := 2.2917604, [96].log_data[42].max := 2.2965894, [96].log_data[42].total := 8259.19, [96].log_data[42].time := 3600.0, [96].log_data[42].minminute := 20, [96].log_data[42].maxminute := 14, [96].log_data[42].valid := 1, [96].log_data[43].min := -0.27999878, [96].log_data[43].max := -0.26000214, [96].log_data[43].total := -986.78827, [96].log_data[43].time := 3600.0, [96].log_data[43].valid := 1, [96].log_data[44].min := -0.30000305, [96].log_data[44].max := -0.30000305, [96].log_data[44].total := -1080.0911, [96].log_data[44].time := 3600.0, [96].log_data[44].valid := 1, [96].log_data[45].time := 3600.0, [96].log_data[45].valid := 1, [96].log_data[46].time := 3600.0, [96].log_data[46].valid := 1, [96].log_data[47].time := 3600.0, [96].log_data[47].valid := 1, [96].log_data[48].min := 6.7492356, [96].log_data[48].max := 6.772595, [96].log_data[48].total := 24320.967, [96].log_data[48].time := 3600.0, [96].log_data[48].minminute := 38, [96].log_data[48].valid := 1, [96].log_data[49].min := 9.188562, [96].log_data[49].max := 9.550131, [96].log_data[49].total := 34143.605, [96].log_data[49].time := 3600.0, [96].log_data[49].maxminute := 53, [96].log_data[49].valid := 1, [96].log_data[50].min := 1.9979122, [96].log_data[50].max := 2.1095629, [96].log_data[50].total := 7398.952, [96].log_data[50].time := 3600.0, [96].log_data[50].minminute := 36, [96].log_data[50].maxminute := 57, [96].log_data[50].valid := 1, [96].log_data[51].time := 3600.0, [96].log_data[51].valid := 1, [96].log_data[52].min := -2.9800034, [96].log_data[52].max := 0.11999512, [96].log_data[52].total := -6705.107, [96].log_data[52].time := 3600.0, [96].log_data[52].minminute := 8, [96].log_data[52].maxminute := 6, [96].log_data[52].valid := 1, [96].log_data[53].min := -2.4800034, [96].log_data[53].max := 0.27999878, [96].log_data[53].total := -6032.156, [96].log_data[53].time := 3600.0, [96].log_data[53].maxminute := 1, [96].log_data[53].valid := 1, [96].log_data[54].max := 0.5405, [96].log_data[54].total := 765.9478, [96].log_data[54].time := 3600.0,
        [96].log_data[54].minminute := 6, [96].log_data[54].maxminute := 8, [96].log_data[54].valid := 1, [96].log_data[55].max := 0.5435, [96].log_data[55].total := 728.5746, [96].log_data[55].time := 3600.0, [96].log_data[55].maxminute := 12, [96].log_data[55].valid := 1, [96].log_data[56].min := 0.15981378, [96].log_data[56].max := 0.16020635, [96].log_data[56].total := 575.90546, [96].log_data[56].time := 3600.0, [96].log_data[56].minminute := 5, [96].log_data[56].maxminute := 28, [96].log_data[56].valid := 1, [96].log_data[57].min := 0.23613189, [96].log_data[57].max := 0.23660298, [96].log_data[57].total := 850.8288, [96].log_data[57].time := 3600.0, [96].log_data[57].minminute := 20, [96].log_data[57].maxminute := 12, [96].log_data[57].valid := 1, [96].log_data[58].time := 3600.0, [96].log_data[58].valid := 1, [96].log_data[59].time := 3600.0, [96].log_data[59].valid := 1, [96].log_data[60].valid := 1, [96].log_data[61].valid := 1, [96].log_data[62].valid := 1, [96].log_data[63].valid := 1, [96].log_data[64].valid := 1, [96].log_data[65].valid := 1, [96].log_data[66].valid := 1, [96].log_data[67].valid := 1, [96].log_data[68].valid := 1, [96].log_data[69].valid := 1, [96].log_data[70].valid := 1, [96].log_data[71].valid := 1, [96].log_data[72].valid := 1, [96].log_data[73].valid := 1, [96].log_data[74].valid := 1, [96].log_data[75].valid := 1, [96].log_data[76].valid := 1, [96].log_data[77].valid := 1, [96].log_data[78].valid := 1, [96].log_data[79].valid := 1, [96].log_data[80].valid := 1, [96].log_data[81].valid := 1, [96].log_data[82].valid := 1, [96].log_data[83].valid := 1, [96].log_data[84].valid := 1, [96].log_data[85].valid := 1, [96].log_data[86].valid := 1, [96].log_data[87].valid := 1, [96].log_data[88].valid := 1, [96].log_data[89].valid := 1, [96].log_data[90].valid := 1, [96].log_data[91].valid := 1, [96].log_data[92].valid := 1, [96].log_data[93].valid := 1,
        [96].log_data[94].valid := 1, [96].log_data[95].valid := 1, [96].log_data[96].valid := 1, [96].log_data[97].valid := 1, [96].log_data[98].valid := 1, [96].log_data[99].valid := 1, [96].log_data[100].valid := 1, [96].log_data[101].valid := 1, [96].log_data[102].valid := 1, [96].log_data[103].valid := 1, [96].log_data[104].valid := 1, [96].log_data[105].valid := 1, [96].log_data[106].valid := 1, [96].log_data[107].valid := 1, [96].log_data[108].valid := 1, [96].log_data[109].valid := 1, [96].log_data[110].valid := 1, [96].log_data[111].valid := 1, [96].log_data[112].valid := 1, [96].log_data[113].valid := 1, [96].log_data[114].valid := 1, [96].log_data[115].valid := 1, [96].log_data[116].valid := 1, [96].log_data[117].valid := 1, [96].log_data[118].valid := 1, [96].log_data[119].valid := 1, [96].log_data[120].valid := 1, [96].log_data[121].valid := 1, [96].log_data[122].valid := 1, [96].log_data[123].valid := 1, [96].log_data[124].valid := 1, [96].time.Year := 2023, [96].time.Month := 1, [96].time.Day := 17, [96].time.Hour := 3, [96].time.Minute := 59, [96].time.Second := 59, [97].log_data[0].min := 1.0, [97].log_data[0].max := 1.0, [97].log_data[0].total := 3600.0, [97].log_data[0].time := 3600.0, [97].log_data[0].valid := 1, [97].log_data[1].time := 3600.0, [97].log_data[1].valid := 1, [97].log_data[2].time := 3600.0, [97].log_data[2].valid := 1, [97].log_data[3].time := 3600.0, [97].log_data[3].valid := 1, [97].log_data[4].time := 3600.0, [97].log_data[4].valid := 1, [97].log_data[5].time := 3600.0, [97].log_data[5].valid := 1, [97].log_data[6].time := 3600.0, [97].log_data[6].valid := 1, [97].log_data[7].time := 3600.0, [97].log_data[7].valid := 1, [97].log_data[8].time := 3600.0, [97].log_data[8].valid := 1, [97].log_data[9].time := 3600.0, [97].log_data[9].valid := 1,
        [97].log_data[10].min := 1.0, [97].log_data[10].max := 1.0, [97].log_data[10].total := 3600.0, [97].log_data[10].time := 3600.0, [97].log_data[10].valid := 1, [97].log_data[11].time := 3600.0, [97].log_data[11].valid := 1, [97].log_data[12].min := 1.0, [97].log_data[12].max := 1.0, [97].log_data[12].total := 3600.0, [97].log_data[12].time := 3600.0, [97].log_data[12].valid := 1, [97].log_data[13].min := 1.0, [97].log_data[13].max := 1.0, [97].log_data[13].total := 3600.0, [97].log_data[13].time := 3600.0, [97].log_data[13].valid := 1, [97].log_data[14].time := 3600.0, [97].log_data[14].valid := 1, [97].log_data[15].time := 3600.0, [97].log_data[15].valid := 1, [97].log_data[16].time := 3600.0, [97].log_data[16].valid := 1, [97].log_data[17].min := 1.0, [97].log_data[17].max := 1.0, [97].log_data[17].total := 3600.0, [97].log_data[17].time := 3600.0, [97].log_data[17].valid := 1, [97].log_data[18].time := 3600.0, [97].log_data[18].valid := 1, [97].log_data[19].time := 3600.0, [97].log_data[19].valid := 1, [97].log_data[20].time := 3600.0, [97].log_data[20].valid := 1, [97].log_data[21].min := 1.0, [97].log_data[21].max := 1.0, [97].log_data[21].total := 3600.0, [97].log_data[21].time := 3600.0, [97].log_data[21].valid := 1, [97].log_data[22].time := 3600.0, [97].log_data[22].valid := 1, [97].log_data[23].time := 3600.0, [97].log_data[23].valid := 1, [97].log_data[24].time := 3600.0, [97].log_data[24].valid := 1, [97].log_data[25].time := 3600.0, [97].log_data[25].valid := 1, [97].log_data[26].time := 3600.0, [97].log_data[26].valid := 1, [97].log_data[27].time := 3600.0, [97].log_data[27].valid := 1, [97].log_data[28].time := 3600.0, [97].log_data[28].valid := 1, [97].log_data[29].min := 1.0, [97].log_data[29].max := 1.0, [97].log_data[29].total := 3600.0, [97].log_data[29].time := 3600.0, [97].log_data[29].valid := 1, [97].log_data[30].min := 1.0, [97].log_data[30].max := 1.0,
        [97].log_data[30].total := 3600.0, [97].log_data[30].time := 3600.0, [97].log_data[30].valid := 1, [97].log_data[31].time := 3600.0, [97].log_data[31].valid := 1, [97].log_data[32].time := 3600.0, [97].log_data[32].valid := 1, [97].log_data[33].time := 3600.0, [97].log_data[33].valid := 1, [97].log_data[34].time := 3600.0, [97].log_data[34].valid := 1, [97].log_data[35].time := 3600.0, [97].log_data[35].valid := 1, [97].log_data[36].time := 3600.0, [97].log_data[36].valid := 1, [97].log_data[37].time := 3600.0, [97].log_data[37].valid := 1, [97].log_data[38].time := 3600.0, [97].log_data[38].valid := 1, [97].log_data[39].min := 0.9935285, [97].log_data[39].max := 1.0045992, [97].log_data[39].total := 3599.1572, [97].log_data[39].time := 3600.0, [97].log_data[39].minminute := 25, [97].log_data[39].maxminute := 15, [97].log_data[39].valid := 1, [97].log_data[40].min := 7.591522, [97].log_data[40].max := 7.603614, [97].log_data[40].total := 27360.857, [97].log_data[40].time := 3600.0, [97].log_data[40].minminute := 20, [97].log_data[40].valid := 1, [97].log_data[41].min := 0.022540038, [97].log_data[41].max := 0.02411035, [97].log_data[41].total := 82.656105, [97].log_data[41].time := 3600.0, [97].log_data[41].minminute := 54, [97].log_data[41].maxminute := 1, [97].log_data[41].valid := 1, [97].log_data[42].min := 2.291525, [97].log_data[42].max := 2.296236, [97].log_data[42].total := 8258.979, [97].log_data[42].time := 3600.0, [97].log_data[42].minminute := 59, [97].log_data[42].maxminute := 6, [97].log_data[42].valid := 1, [97].log_data[43].min := -0.27999878, [97].log_data[43].max := -0.26000214, [97].log_data[43].total := -970.6451, [97].log_data[43].time := 3600.0, [97].log_data[43].valid := 1, [97].log_data[44].min := -0.30000305, [97].log_data[44].max := -0.30000305, [97].log_data[44].total := -1080.0911, [97].log_data[44].time := 3600.0, [97].log_data[44].valid := 1, [97].log_data[45].time := 3600.0, [97].log_data[45].valid := 1, [97].log_data[46].time := 3600.0, [97].log_data[46].valid := 1,
        [97].log_data[47].time := 3600.0, [97].log_data[47].valid := 1, [97].log_data[48].min := 6.7550073, [97].log_data[48].max := 6.77287, [97].log_data[48].total := 24353.275, [97].log_data[48].time := 3600.0, [97].log_data[48].maxminute := 58, [97].log_data[48].valid := 1, [97].log_data[49].min := 9.510088, [97].log_data[49].max := 9.581735, [97].log_data[49].total := 34368.902, [97].log_data[49].time := 3600.0, [97].log_data[49].maxminute := 55, [97].log_data[49].valid := 1, [97].log_data[50].min := 2.1034384, [97].log_data[50].max := 2.1145093, [97].log_data[50].total := 7598.7866, [97].log_data[50].time := 3600.0, [97].log_data[50].minminute := 1, [97].log_data[50].maxminute := 59, [97].log_data[50].valid := 1, [97].log_data[51].time := 3600.0, [97].log_data[51].valid := 1, [97].log_data[52].min := -1.6600037, [97].log_data[52].max := -1.4400024, [97].log_data[52].total := -5550.623, [97].log_data[52].time := 3600.0, [97].log_data[52].minminute := 59, [97].log_data[52].maxminute := 5, [97].log_data[52].valid := 1, [97].log_data[53].min := -1.4800034, [97].log_data[53].max := -1.300003, [97].log_data[53].total := -5051.91, [97].log_data[53].time := 3600.0, [97].log_data[53].minminute := 15, [97].log_data[53].maxminute := 5, [97].log_data[53].valid := 1, [97].log_data[54].time := 3600.0, [97].log_data[54].valid := 1, [97].log_data[55].time := 3600.0, [97].log_data[55].valid := 1, [97].log_data[56].min := 0.15977451, [97].log_data[56].max := 0.16020635, [97].log_data[56].total := 575.8309, [97].log_data[56].time := 3600.0, [97].log_data[56].minminute := 44, [97].log_data[56].maxminute := 19, [97].log_data[56].valid := 1, [97].log_data[57].min := 0.23617114, [97].log_data[57].max := 0.23660298, [97].log_data[57].total := 850.8692, [97].log_data[57].time := 3600.0, [97].log_data[57].minminute := 10, [97].log_data[57].maxminute := 25, [97].log_data[57].valid := 1, [97].log_data[58].time := 3600.0, [97].log_data[58].valid := 1, [97].log_data[59].time := 3600.0, [97].log_data[59].valid := 1, [97].log_data[60].valid := 1,
        [97].log_data[61].valid := 1, [97].log_data[62].valid := 1, [97].log_data[63].valid := 1, [97].log_data[64].valid := 1, [97].log_data[65].valid := 1, [97].log_data[66].valid := 1, [97].log_data[67].valid := 1, [97].log_data[68].valid := 1, [97].log_data[69].valid := 1, [97].log_data[70].valid := 1, [97].log_data[71].valid := 1, [97].log_data[72].valid := 1, [97].log_data[73].valid := 1, [97].log_data[74].valid := 1, [97].log_data[75].valid := 1, [97].log_data[76].valid := 1, [97].log_data[77].valid := 1, [97].log_data[78].valid := 1, [97].log_data[79].valid := 1, [97].log_data[80].valid := 1, [97].log_data[81].valid := 1, [97].log_data[82].valid := 1, [97].log_data[83].valid := 1, [97].log_data[84].valid := 1, [97].log_data[85].valid := 1, [97].log_data[86].valid := 1, [97].log_data[87].valid := 1, [97].log_data[88].valid := 1, [97].log_data[89].valid := 1, [97].log_data[90].valid := 1, [97].log_data[91].valid := 1, [97].log_data[92].valid := 1, [97].log_data[93].valid := 1, [97].log_data[94].valid := 1, [97].log_data[95].valid := 1, [97].log_data[96].valid := 1, [97].log_data[97].valid := 1, [97].log_data[98].valid := 1, [97].log_data[99].valid := 1, [97].log_data[100].valid := 1, [97].log_data[101].valid := 1, [97].log_data[102].valid := 1, [97].log_data[103].valid := 1, [97].log_data[104].valid := 1, [97].log_data[105].valid := 1, [97].log_data[106].valid := 1, [97].log_data[107].valid := 1, [97].log_data[108].valid := 1, [97].log_data[109].valid := 1, [97].log_data[110].valid := 1, [97].log_data[111].valid := 1, [97].log_data[112].valid := 1, [97].log_data[113].valid := 1, [97].log_data[114].valid := 1, [97].log_data[115].valid := 1, [97].log_data[116].valid := 1, [97].log_data[117].valid := 1, [97].log_data[118].valid := 1, [97].log_data[119].valid := 1, [97].log_data[120].valid := 1,
        [97].log_data[121].valid := 1, [97].log_data[122].valid := 1, [97].log_data[123].valid := 1, [97].log_data[124].valid := 1, [97].time.Year := 2023, [97].time.Month := 1, [97].time.Day := 17, [97].time.Hour := 4, [97].time.Minute := 59, [97].time.Second := 59, [98].log_data[0].min := 1.0, [98].log_data[0].max := 1.0, [98].log_data[0].total := 3600.0, [98].log_data[0].time := 3600.0, [98].log_data[0].valid := 1, [98].log_data[1].time := 3600.0, [98].log_data[1].valid := 1, [98].log_data[2].time := 3600.0, [98].log_data[2].valid := 1, [98].log_data[3].time := 3600.0, [98].log_data[3].valid := 1, [98].log_data[4].time := 3600.0, [98].log_data[4].valid := 1, [98].log_data[5].time := 3600.0, [98].log_data[5].valid := 1, [98].log_data[6].time := 3600.0, [98].log_data[6].valid := 1, [98].log_data[7].time := 3600.0, [98].log_data[7].valid := 1, [98].log_data[8].time := 3600.0, [98].log_data[8].valid := 1, [98].log_data[9].time := 3600.0, [98].log_data[9].valid := 1, [98].log_data[10].min := 1.0, [98].log_data[10].max := 1.0, [98].log_data[10].total := 3600.0, [98].log_data[10].time := 3600.0, [98].log_data[10].valid := 1, [98].log_data[11].time := 3600.0, [98].log_data[11].valid := 1, [98].log_data[12].min := 1.0, [98].log_data[12].max := 1.0, [98].log_data[12].total := 3600.0, [98].log_data[12].time := 3600.0, [98].log_data[12].valid := 1, [98].log_data[13].min := 1.0, [98].log_data[13].max := 1.0, [98].log_data[13].total := 3600.0, [98].log_data[13].time := 3600.0, [98].log_data[13].valid := 1, [98].log_data[14].time := 3600.0, [98].log_data[14].valid := 1, [98].log_data[15].time := 3600.0, [98].log_data[15].valid := 1, [98].log_data[16].time := 3600.0, [98].log_data[16].valid := 1, [98].log_data[17].min := 1.0, [98].log_data[17].max := 1.0, [98].log_data[17].total := 3600.0, [98].log_data[17].time := 3600.0,
        [98].log_data[17].valid := 1, [98].log_data[18].time := 3600.0, [98].log_data[18].valid := 1, [98].log_data[19].time := 3600.0, [98].log_data[19].valid := 1, [98].log_data[20].time := 3600.0, [98].log_data[20].valid := 1, [98].log_data[21].min := 1.0, [98].log_data[21].max := 1.0, [98].log_data[21].total := 3600.0, [98].log_data[21].time := 3600.0, [98].log_data[21].valid := 1, [98].log_data[22].time := 3600.0, [98].log_data[22].valid := 1, [98].log_data[23].time := 3600.0, [98].log_data[23].valid := 1, [98].log_data[24].time := 3600.0, [98].log_data[24].valid := 1, [98].log_data[25].time := 3600.0, [98].log_data[25].valid := 1, [98].log_data[26].time := 3600.0, [98].log_data[26].valid := 1, [98].log_data[27].time := 3600.0, [98].log_data[27].valid := 1, [98].log_data[28].time := 3600.0, [98].log_data[28].valid := 1, [98].log_data[29].min := 1.0, [98].log_data[29].max := 1.0, [98].log_data[29].total := 3600.0, [98].log_data[29].time := 3600.0, [98].log_data[29].valid := 1, [98].log_data[30].min := 1.0, [98].log_data[30].max := 1.0, [98].log_data[30].total := 3600.0, [98].log_data[30].time := 3600.0, [98].log_data[30].valid := 1, [98].log_data[31].time := 3600.0, [98].log_data[31].valid := 1, [98].log_data[32].time := 3600.0, [98].log_data[32].valid := 1, [98].log_data[33].time := 3600.0, [98].log_data[33].valid := 1, [98].log_data[34].time := 3600.0, [98].log_data[34].valid := 1, [98].log_data[35].time := 3600.0, [98].log_data[35].valid := 1, [98].log_data[36].time := 3600.0, [98].log_data[36].valid := 1, [98].log_data[37].time := 3600.0, [98].log_data[37].valid := 1, [98].log_data[38].time := 3600.0, [98].log_data[38].valid := 1, [98].log_data[39].min := 0.99435294, [98].log_data[39].max := 1.0037748, [98].log_data[39].total := 3598.5107, [98].log_data[39].time := 3600.0, [98].log_data[39].maxminute := 51, [98].log_data[39].valid := 1, [98].log_data[40].min := 7.5942707, [98].log_data[40].max := 7.603614,
        [98].log_data[40].total := 27361.576, [98].log_data[40].time := 3600.0, [98].log_data[40].minminute := 39, [98].log_data[40].maxminute := 42, [98].log_data[40].valid := 1, [98].log_data[41].min := 0.02273633, [98].log_data[41].max := 0.030195557, [98].log_data[41].total := 84.19409, [98].log_data[41].time := 3600.0, [98].log_data[41].maxminute := 49, [98].log_data[41].valid := 1, [98].log_data[42].min := 2.2917604, [98].log_data[42].max := 2.296236, [98].log_data[42].total := 8258.938, [98].log_data[42].time := 3600.0, [98].log_data[42].minminute := 26, [98].log_data[42].maxminute := 14, [98].log_data[42].valid := 1, [98].log_data[43].min := -0.27999878, [98].log_data[43].max := -0.26000214, [98].log_data[43].total := -993.7968, [98].log_data[43].time := 3600.0, [98].log_data[43].valid := 1, [98].log_data[44].min := -0.30000305, [98].log_data[44].max := -0.30000305, [98].log_data[44].total := -1080.0911, [98].log_data[44].time := 3600.0, [98].log_data[44].valid := 1, [98].log_data[45].time := 3600.0, [98].log_data[45].valid := 1, [98].log_data[46].time := 3600.0, [98].log_data[46].valid := 1, [98].log_data[47].time := 3600.0, [98].log_data[47].valid := 1, [98].log_data[48].min := 6.7706714, [98].log_data[48].max := 6.782763, [98].log_data[48].total := 24394.18, [98].log_data[48].time := 3600.0, [98].log_data[48].maxminute := 58, [98].log_data[48].valid := 1, [98].log_data[49].min := 9.545617, [98].log_data[49].max := 9.611177, [98].log_data[49].total := 34496.05, [98].log_data[49].time := 3600.0, [98].log_data[49].minminute := 3, [98].log_data[49].maxminute := 50, [98].log_data[49].valid := 1, [98].log_data[50].min := 2.106854, [98].log_data[50].max := 2.1154513, [98].log_data[50].total := 7606.2656, [98].log_data[50].time := 3600.0, [98].log_data[50].minminute := 13, [98].log_data[50].maxminute := 36, [98].log_data[50].valid := 1, [98].log_data[51].time := 3600.0, [98].log_data[51].valid := 1, [98].log_data[52].min := -1.6800003, [98].log_data[52].max := -1.4800034, [98].log_data[52].total := -5682.6035, [98].log_data[52].time := 3600.0,
        [98].log_data[52].minminute := 33, [98].log_data[52].valid := 1, [98].log_data[53].min := -1.5200043, [98].log_data[53].max := -1.340004, [98].log_data[53].total := -5124.765, [98].log_data[53].time := 3600.0, [98].log_data[53].minminute := 33, [98].log_data[53].valid := 1, [98].log_data[54].time := 3600.0, [98].log_data[54].valid := 1, [98].log_data[55].time := 3600.0, [98].log_data[55].valid := 1, [98].log_data[56].min := 0.159696, [98].log_data[56].max := 0.16016708, [98].log_data[56].total := 575.68146, [98].log_data[56].time := 3600.0, [98].log_data[56].minminute := 20, [98].log_data[56].maxminute := 39, [98].log_data[56].valid := 1, [98].log_data[57].min := 0.2362104, [98].log_data[57].max := 0.23660298, [98].log_data[57].total := 850.9017, [98].log_data[57].time := 3600.0, [98].log_data[57].minminute := 9, [98].log_data[57].maxminute := 3, [98].log_data[57].valid := 1, [98].log_data[58].time := 3600.0, [98].log_data[58].valid := 1, [98].log_data[59].time := 3600.0, [98].log_data[59].valid := 1, [98].log_data[60].valid := 1, [98].log_data[61].valid := 1, [98].log_data[62].valid := 1, [98].log_data[63].valid := 1, [98].log_data[64].valid := 1, [98].log_data[65].valid := 1, [98].log_data[66].valid := 1, [98].log_data[67].valid := 1, [98].log_data[68].valid := 1, [98].log_data[69].valid := 1, [98].log_data[70].valid := 1, [98].log_data[71].valid := 1, [98].log_data[72].valid := 1, [98].log_data[73].valid := 1, [98].log_data[74].valid := 1, [98].log_data[75].valid := 1, [98].log_data[76].valid := 1, [98].log_data[77].valid := 1, [98].log_data[78].valid := 1, [98].log_data[79].valid := 1, [98].log_data[80].valid := 1, [98].log_data[81].valid := 1, [98].log_data[82].valid := 1, [98].log_data[83].valid := 1, [98].log_data[84].valid := 1, [98].log_data[85].valid := 1, [98].log_data[86].valid := 1, [98].log_data[87].valid := 1, [98].log_data[88].valid := 1, [98].log_data[89].valid := 1,
        [98].log_data[90].valid := 1, [98].log_data[91].valid := 1, [98].log_data[92].valid := 1, [98].log_data[93].valid := 1, [98].log_data[94].valid := 1, [98].log_data[95].valid := 1, [98].log_data[96].valid := 1, [98].log_data[97].valid := 1, [98].log_data[98].valid := 1, [98].log_data[99].valid := 1, [98].log_data[100].valid := 1, [98].log_data[101].valid := 1, [98].log_data[102].valid := 1, [98].log_data[103].valid := 1, [98].log_data[104].valid := 1, [98].log_data[105].valid := 1, [98].log_data[106].valid := 1, [98].log_data[107].valid := 1, [98].log_data[108].valid := 1, [98].log_data[109].valid := 1, [98].log_data[110].valid := 1, [98].log_data[111].valid := 1, [98].log_data[112].valid := 1, [98].log_data[113].valid := 1, [98].log_data[114].valid := 1, [98].log_data[115].valid := 1, [98].log_data[116].valid := 1, [98].log_data[117].valid := 1, [98].log_data[118].valid := 1, [98].log_data[119].valid := 1, [98].log_data[120].valid := 1, [98].log_data[121].valid := 1, [98].log_data[122].valid := 1, [98].log_data[123].valid := 1, [98].log_data[124].valid := 1, [98].time.Year := 2023, [98].time.Month := 1, [98].time.Day := 17, [98].time.Hour := 5, [98].time.Minute := 59, [98].time.Second := 59, [99].log_data[0].min := 1.0, [99].log_data[0].max := 1.0, [99].log_data[0].total := 3600.0, [99].log_data[0].time := 3600.0, [99].log_data[0].valid := 1, [99].log_data[1].max := 1.0, [99].log_data[1].total := 541.0, [99].log_data[1].time := 3600.0, [99].log_data[1].maxminute := 43, [99].log_data[1].valid := 1, [99].log_data[2].max := 1.0, [99].log_data[2].total := 537.5, [99].log_data[2].time := 3600.0, [99].log_data[2].maxminute := 44, [99].log_data[2].valid := 1, [99].log_data[3].time := 3600.0, [99].log_data[3].valid := 1, [99].log_data[4].time := 3600.0, [99].log_data[4].valid := 1,
        [99].log_data[5].max := 1.0, [99].log_data[5].total := 223.0, [99].log_data[5].time := 3600.0, [99].log_data[5].maxminute := 46, [99].log_data[5].valid := 1, [99].log_data[6].time := 3600.0, [99].log_data[6].valid := 1, [99].log_data[7].time := 3600.0, [99].log_data[7].valid := 1, [99].log_data[8].max := 1.0, [99].log_data[8].total := 707.249, [99].log_data[8].time := 3600.0, [99].log_data[8].maxminute := 48, [99].log_data[8].valid := 1, [99].log_data[9].max := 1.0, [99].log_data[9].total := 703.749, [99].log_data[9].time := 3600.0, [99].log_data[9].maxminute := 48, [99].log_data[9].valid := 1, [99].log_data[10].min := 1.0, [99].log_data[10].max := 1.0, [99].log_data[10].total := 3600.0, [99].log_data[10].time := 3600.0, [99].log_data[10].valid := 1, [99].log_data[11].time := 3600.0, [99].log_data[11].valid := 1, [99].log_data[12].min := 1.0, [99].log_data[12].max := 1.0, [99].log_data[12].total := 3600.0, [99].log_data[12].time := 3600.0, [99].log_data[12].valid := 1, [99].log_data[13].min := 1.0, [99].log_data[13].max := 1.0, [99].log_data[13].total := 3600.0, [99].log_data[13].time := 3600.0, [99].log_data[13].valid := 1, [99].log_data[14].time := 3600.0, [99].log_data[14].valid := 1, [99].log_data[15].time := 3600.0, [99].log_data[15].valid := 1, [99].log_data[16].time := 3600.0, [99].log_data[16].valid := 1, [99].log_data[17].min := 1.0, [99].log_data[17].max := 1.0, [99].log_data[17].total := 3600.0, [99].log_data[17].time := 3600.0, [99].log_data[17].valid := 1, [99].log_data[18].time := 3600.0, [99].log_data[18].valid := 1, [99].log_data[19].time := 3600.0, [99].log_data[19].valid := 1, [99].log_data[20].time := 3600.0, [99].log_data[20].valid := 1, [99].log_data[21].min := 1.0, [99].log_data[21].max := 1.0, [99].log_data[21].total := 3600.0, [99].log_data[21].time := 3600.0, [99].log_data[21].valid := 1, [99].log_data[22].time := 3600.0, [99].log_data[22].valid := 1,
        [99].log_data[23].time := 3600.0, [99].log_data[23].valid := 1, [99].log_data[24].time := 3600.0, [99].log_data[24].valid := 1, [99].log_data[25].time := 3600.0, [99].log_data[25].valid := 1, [99].log_data[26].time := 3600.0, [99].log_data[26].valid := 1, [99].log_data[27].time := 3600.0, [99].log_data[27].valid := 1, [99].log_data[28].time := 3600.0, [99].log_data[28].valid := 1, [99].log_data[29].min := 1.0, [99].log_data[29].max := 1.0, [99].log_data[29].total := 3600.0, [99].log_data[29].time := 3600.0, [99].log_data[29].valid := 1, [99].log_data[30].min := 1.0, [99].log_data[30].max := 1.0, [99].log_data[30].total := 3600.0, [99].log_data[30].time := 3600.0, [99].log_data[30].valid := 1, [99].log_data[31].max := 1.0, [99].log_data[31].total := 501.249, [99].log_data[31].time := 3600.0, [99].log_data[31].maxminute := 51, [99].log_data[31].valid := 1, [99].log_data[32].max := 1.0, [99].log_data[32].total := 110.749, [99].log_data[32].time := 3600.0, [99].log_data[32].maxminute := 48, [99].log_data[32].valid := 1, [99].log_data[33].time := 3600.0, [99].log_data[33].valid := 1, [99].log_data[34].time := 3600.0, [99].log_data[34].valid := 1, [99].log_data[35].max := 1.0, [99].log_data[35].total := 238.249, [99].log_data[35].time := 3600.0, [99].log_data[35].maxminute := 56, [99].log_data[35].valid := 1, [99].log_data[36].max := 1.0, [99].log_data[36].total := 370.249, [99].log_data[36].time := 3600.0, [99].log_data[36].maxminute := 48, [99].log_data[36].valid := 1, [99].log_data[37].max := 7.263107, [99].log_data[37].total := 3397.304, [99].log_data[37].time := 3600.0, [99].log_data[37].maxminute := 44, [99].log_data[37].valid := 1, [99].log_data[38].time := 3600.0, [99].log_data[38].valid := 1, [99].log_data[39].min := 0.9947063, [99].log_data[39].max := 1.0212055, [99].log_data[39].total := 3604.9814, [99].log_data[39].time := 3600.0, [99].log_data[39].maxminute := 46, [99].log_data[39].valid := 1, [99].log_data[40].min := 7.5959196,
        [99].log_data[40].max := 7.60224, [99].log_data[40].total := 27362.14, [99].log_data[40].time := 3600.0, [99].log_data[40].minminute := 57, [99].log_data[40].valid := 1, [99].log_data[41].min := 0.02273633, [99].log_data[41].max := 0.02411035, [99].log_data[41].total := 82.598595, [99].log_data[41].time := 3600.0, [99].log_data[41].maxminute := 21, [99].log_data[41].valid := 1, [99].log_data[42].min := 2.291407, [99].log_data[42].max := 2.2963536, [99].log_data[42].total := 8258.93, [99].log_data[42].time := 3600.0, [99].log_data[42].minminute := 24, [99].log_data[42].maxminute := 25, [99].log_data[42].valid := 1, [99].log_data[43].min := -0.27999878, [99].log_data[43].max := -0.26000214, [99].log_data[43].total := -1006.2909, [99].log_data[43].time := 3600.0, [99].log_data[43].valid := 1, [99].log_data[44].min := -0.3199997, [99].log_data[44].max := -0.30000305, [99].log_data[44].total := -1080.7041, [99].log_data[44].time := 3600.0, [99].log_data[44].minminute := 26, [99].log_data[44].valid := 1, [99].log_data[45].time := 3600.0, [99].log_data[45].valid := 1, [99].log_data[46].time := 3600.0, [99].log_data[46].valid := 1, [99].log_data[47].time := 3600.0, [99].log_data[47].valid := 1, [99].log_data[48].min := 6.749511, [99].log_data[48].max := 6.9765024, [99].log_data[48].total := 24476.17, [99].log_data[48].time := 3600.0, [99].log_data[48].minminute := 59, [99].log_data[48].maxminute := 53, [99].log_data[48].valid := 1, [99].log_data[49].min := 7.8206086, [99].log_data[49].max := 9.639443, [99].log_data[49].total := 33926.59, [99].log_data[49].time := 3600.0, [99].log_data[49].minminute := 59, [99].log_data[49].maxminute := 46, [99].log_data[49].valid := 1, [99].log_data[50].min := 2.0679882, [99].log_data[50].max := 2.150784, [99].log_data[50].total := 7602.42, [99].log_data[50].time := 3600.0, [99].log_data[50].minminute := 51, [99].log_data[50].maxminute := 48, [99].log_data[50].valid := 1, [99].log_data[51].time := 3600.0, [99].log_data[51].valid := 1, [99].log_data[52].min := -4.220001, [99].log_data[52].max := 0.11999512,
        [99].log_data[52].total := -6199.435, [99].log_data[52].time := 3600.0, [99].log_data[52].minminute := 48, [99].log_data[52].maxminute := 50, [99].log_data[52].valid := 1, [99].log_data[53].min := -3.899994, [99].log_data[53].max := 0.27999878, [99].log_data[53].total := -5576.114, [99].log_data[53].time := 3600.0, [99].log_data[53].minminute := 48, [99].log_data[53].maxminute := 55, [99].log_data[53].valid := 1, [99].log_data[54].max := 0.51199996, [99].log_data[54].total := 240.80893, [99].log_data[54].time := 3600.0, [99].log_data[54].maxminute := 51, [99].log_data[54].valid := 1, [99].log_data[55].max := 0.502, [99].log_data[55].total := 239.22891, [99].log_data[55].time := 3600.0, [99].log_data[55].maxminute := 56, [99].log_data[55].valid := 1, [99].log_data[56].min := 0.159696, [99].log_data[56].max := 0.16012783, [99].log_data[56].total := 575.5295, [99].log_data[56].time := 3600.0, [99].log_data[56].minminute := 25, [99].log_data[56].valid := 1, [99].log_data[57].min := 0.23613189, [99].log_data[57].max := 0.23660298, [99].log_data[57].total := 850.8992, [99].log_data[57].time := 3600.0, [99].log_data[57].minminute := 50, [99].log_data[57].maxminute := 7, [99].log_data[57].valid := 1, [99].log_data[58].time := 3600.0, [99].log_data[58].valid := 1, [99].log_data[59].time := 3600.0, [99].log_data[59].valid := 1, [99].log_data[60].valid := 1, [99].log_data[61].valid := 1, [99].log_data[62].valid := 1, [99].log_data[63].valid := 1, [99].log_data[64].valid := 1, [99].log_data[65].valid := 1, [99].log_data[66].valid := 1, [99].log_data[67].valid := 1, [99].log_data[68].valid := 1, [99].log_data[69].valid := 1, [99].log_data[70].valid := 1, [99].log_data[71].valid := 1, [99].log_data[72].valid := 1, [99].log_data[73].valid := 1, [99].log_data[74].valid := 1, [99].log_data[75].valid := 1, [99].log_data[76].valid := 1, [99].log_data[77].valid := 1, [99].log_data[78].valid := 1, [99].log_data[79].valid := 1, [99].log_data[80].valid := 1,
        [99].log_data[81].valid := 1, [99].log_data[82].valid := 1, [99].log_data[83].valid := 1, [99].log_data[84].valid := 1, [99].log_data[85].valid := 1, [99].log_data[86].valid := 1, [99].log_data[87].valid := 1, [99].log_data[88].valid := 1, [99].log_data[89].valid := 1, [99].log_data[90].valid := 1, [99].log_data[91].valid := 1, [99].log_data[92].valid := 1, [99].log_data[93].valid := 1, [99].log_data[94].valid := 1, [99].log_data[95].valid := 1, [99].log_data[96].valid := 1, [99].log_data[97].valid := 1, [99].log_data[98].valid := 1, [99].log_data[99].valid := 1, [99].log_data[100].valid := 1, [99].log_data[101].valid := 1, [99].log_data[102].valid := 1, [99].log_data[103].valid := 1, [99].log_data[104].valid := 1, [99].log_data[105].valid := 1, [99].log_data[106].valid := 1, [99].log_data[107].valid := 1, [99].log_data[108].valid := 1, [99].log_data[109].valid := 1, [99].log_data[110].valid := 1, [99].log_data[111].valid := 1, [99].log_data[112].valid := 1, [99].log_data[113].valid := 1, [99].log_data[114].valid := 1, [99].log_data[115].valid := 1, [99].log_data[116].valid := 1, [99].log_data[117].valid := 1, [99].log_data[118].valid := 1, [99].log_data[119].valid := 1, [99].log_data[120].valid := 1, [99].log_data[121].valid := 1, [99].log_data[122].valid := 1, [99].log_data[123].valid := 1, [99].log_data[124].valid := 1, [99].time.Year := 2023, [99].time.Month := 1, [99].time.Day := 17, [99].time.Hour := 6, [99].time.Minute := 59, [99].time.Second := 59, [100].log_data[0].min := 1.0, [100].log_data[0].max := 1.0, [100].log_data[0].total := 3600.0, [100].log_data[0].time := 3600.0, [100].log_data[0].valid := 1, [100].log_data[1].time := 3600.0, [100].log_data[1].valid := 1, [100].log_data[2].time := 3600.0, [100].log_data[2].valid := 1, [100].log_data[3].time := 3600.0,
        [100].log_data[3].valid := 1, [100].log_data[4].time := 3600.0, [100].log_data[4].valid := 1, [100].log_data[5].time := 3600.0, [100].log_data[5].valid := 1, [100].log_data[6].time := 3600.0, [100].log_data[6].valid := 1, [100].log_data[7].time := 3600.0, [100].log_data[7].valid := 1, [100].log_data[8].min := 1.0, [100].log_data[8].max := 1.0, [100].log_data[8].total := 3600.0, [100].log_data[8].time := 3600.0, [100].log_data[8].valid := 1, [100].log_data[9].min := 1.0, [100].log_data[9].max := 1.0, [100].log_data[9].total := 3600.0, [100].log_data[9].time := 3600.0, [100].log_data[9].valid := 1, [100].log_data[10].min := 1.0, [100].log_data[10].max := 1.0, [100].log_data[10].total := 3600.0, [100].log_data[10].time := 3600.0, [100].log_data[10].valid := 1, [100].log_data[11].time := 3600.0, [100].log_data[11].valid := 1, [100].log_data[12].min := 1.0, [100].log_data[12].max := 1.0, [100].log_data[12].total := 3600.0, [100].log_data[12].time := 3600.0, [100].log_data[12].valid := 1, [100].log_data[13].min := 1.0, [100].log_data[13].max := 1.0, [100].log_data[13].total := 3600.0, [100].log_data[13].time := 3600.0, [100].log_data[13].valid := 1, [100].log_data[14].time := 3600.0, [100].log_data[14].valid := 1, [100].log_data[15].time := 3600.0, [100].log_data[15].valid := 1, [100].log_data[16].time := 3600.0, [100].log_data[16].valid := 1, [100].log_data[17].min := 1.0, [100].log_data[17].max := 1.0, [100].log_data[17].total := 3600.0, [100].log_data[17].time := 3600.0, [100].log_data[17].valid := 1, [100].log_data[18].time := 3600.0, [100].log_data[18].valid := 1, [100].log_data[19].time := 3600.0, [100].log_data[19].valid := 1, [100].log_data[20].time := 3600.0, [100].log_data[20].valid := 1, [100].log_data[21].min := 1.0, [100].log_data[21].max := 1.0, [100].log_data[21].total := 3600.0, [100].log_data[21].time := 3600.0, [100].log_data[21].valid := 1, [100].log_data[22].time := 3600.0, [100].log_data[22].valid := 1,
        [100].log_data[23].time := 3600.0, [100].log_data[23].valid := 1, [100].log_data[24].time := 3600.0, [100].log_data[24].valid := 1, [100].log_data[25].time := 3600.0, [100].log_data[25].valid := 1, [100].log_data[26].time := 3600.0, [100].log_data[26].valid := 1, [100].log_data[27].time := 3600.0, [100].log_data[27].valid := 1, [100].log_data[28].time := 3600.0, [100].log_data[28].valid := 1, [100].log_data[29].min := 1.0, [100].log_data[29].max := 1.0, [100].log_data[29].total := 3600.0, [100].log_data[29].time := 3600.0, [100].log_data[29].valid := 1, [100].log_data[30].min := 1.0, [100].log_data[30].max := 1.0, [100].log_data[30].total := 3600.0, [100].log_data[30].time := 3600.0, [100].log_data[30].valid := 1, [100].log_data[31].max := 1.0, [100].log_data[31].total := 1440.998, [100].log_data[31].time := 3600.0, [100].log_data[31].valid := 1, [100].log_data[32].max := 1.0, [100].log_data[32].total := 1629.998, [100].log_data[32].time := 3600.0, [100].log_data[32].maxminute := 2, [100].log_data[32].valid := 1, [100].log_data[33].time := 3600.0, [100].log_data[33].valid := 1, [100].log_data[34].time := 3600.0, [100].log_data[34].valid := 1, [100].log_data[35].max := 1.0, [100].log_data[35].total := 1440.249, [100].log_data[35].time := 3600.0, [100].log_data[35].minminute := 5, [100].log_data[35].valid := 1, [100].log_data[36].max := 1.0, [100].log_data[36].total := 1629.7471, [100].log_data[36].time := 3600.0, [100].log_data[36].maxminute := 6, [100].log_data[36].valid := 1, [100].log_data[37].time := 3600.0, [100].log_data[37].valid := 1, [100].log_data[38].time := 3600.0, [100].log_data[38].valid := 1, [100].log_data[39].min := 0.9936463, [100].log_data[39].max := 1.0055416, [100].log_data[39].total := 3603.9526, [100].log_data[39].time := 3600.0, [100].log_data[39].minminute := 48, [100].log_data[39].maxminute := 29, [100].log_data[39].valid := 1, [100].log_data[40].min := 7.5942707, [100].log_data[40].max := 7.603614, [100].log_data[40].total := 27362.895, [100].log_data[40].time := 3600.0,
        [100].log_data[40].minminute := 4, [100].log_data[40].maxminute := 6, [100].log_data[40].valid := 1, [100].log_data[41].min := 0.02273633, [100].log_data[41].max := 0.02411035, [100].log_data[41].total := 82.52954, [100].log_data[41].time := 3600.0, [100].log_data[41].valid := 1, [100].log_data[42].min := 2.290936, [100].log_data[42].max := 2.296118, [100].log_data[42].total := 8258.949, [100].log_data[42].time := 3600.0, [100].log_data[42].minminute := 12, [100].log_data[42].maxminute := 52, [100].log_data[42].valid := 1, [100].log_data[43].min := -0.27999878, [100].log_data[43].max := -0.26000214, [100].log_data[43].total := -1007.19446, [100].log_data[43].time := 3600.0, [100].log_data[43].maxminute := 17, [100].log_data[43].valid := 1, [100].log_data[44].min := -0.3199997, [100].log_data[44].max := -0.30000305, [100].log_data[44].total := -1083.5392, [100].log_data[44].time := 3600.0, [100].log_data[44].valid := 1, [100].log_data[45].time := 3600.0, [100].log_data[45].valid := 1, [100].log_data[46].time := 3600.0, [100].log_data[46].valid := 1, [100].log_data[47].time := 3600.0, [100].log_data[47].valid := 1, [100].log_data[48].min := 6.5923214, [100].log_data[48].max := 6.7981515, [100].log_data[48].total := 24189.898, [100].log_data[48].time := 3600.0, [100].log_data[48].minminute := 18, [100].log_data[48].maxminute := 32, [100].log_data[48].valid := 1, [100].log_data[49].min := 6.9902954, [100].log_data[49].max := 9.478878, [100].log_data[49].total := 30073.879, [100].log_data[49].time := 3600.0, [100].log_data[49].minminute := 14, [100].log_data[49].maxminute := 58, [100].log_data[49].valid := 1, [100].log_data[50].min := 2.0201716, [100].log_data[50].max := 2.1039095, [100].log_data[50].total := 7424.4717, [100].log_data[50].time := 3600.0, [100].log_data[50].minminute := 59, [100].log_data[50].valid := 1, [100].log_data[51].time := 3600.0, [100].log_data[51].valid := 1, [100].log_data[52].min := -3.0999985, [100].log_data[52].max := 0.11999512, [100].log_data[52].total := -7586.4966, [100].log_data[52].time := 3600.0, [100].log_data[52].minminute := 12, [100].log_data[52].valid := 1,
        [100].log_data[53].min := -2.4600067, [100].log_data[53].max := 0.30000305, [100].log_data[53].total := -6896.288, [100].log_data[53].time := 3600.0, [100].log_data[53].minminute := 21, [100].log_data[53].maxminute := 27, [100].log_data[53].valid := 1, [100].log_data[54].max := 0.554, [100].log_data[54].total := 1217.3843, [100].log_data[54].time := 3600.0, [100].log_data[54].maxminute := 12, [100].log_data[54].valid := 1, [100].log_data[55].max := 0.51350003, [100].log_data[55].total := 1216.7537, [100].log_data[55].time := 3600.0, [100].log_data[55].minminute := 5, [100].log_data[55].maxminute := 17, [100].log_data[55].valid := 1, [100].log_data[56].min := 0.15957822, [100].log_data[56].max := 0.16008857, [100].log_data[56].total := 575.34424, [100].log_data[56].time := 3600.0, [100].log_data[56].minminute := 24, [100].log_data[56].maxminute := 10, [100].log_data[56].valid := 1, [100].log_data[57].min := 0.23440449, [100].log_data[57].max := 0.23660298, [100].log_data[57].total := 846.76575, [100].log_data[57].time := 3600.0, [100].log_data[57].minminute := 50, [100].log_data[57].maxminute := 5, [100].log_data[57].valid := 1, [100].log_data[58].time := 3600.0, [100].log_data[58].valid := 1, [100].log_data[59].time := 3600.0, [100].log_data[59].valid := 1, [100].log_data[60].valid := 1, [100].log_data[61].valid := 1, [100].log_data[62].valid := 1, [100].log_data[63].valid := 1, [100].log_data[64].valid := 1, [100].log_data[65].valid := 1, [100].log_data[66].valid := 1, [100].log_data[67].valid := 1, [100].log_data[68].valid := 1, [100].log_data[69].valid := 1, [100].log_data[70].valid := 1, [100].log_data[71].valid := 1, [100].log_data[72].valid := 1, [100].log_data[73].valid := 1, [100].log_data[74].valid := 1, [100].log_data[75].valid := 1, [100].log_data[76].valid := 1, [100].log_data[77].valid := 1, [100].log_data[78].valid := 1, [100].log_data[79].valid := 1, [100].log_data[80].valid := 1, [100].log_data[81].valid := 1, [100].log_data[82].valid := 1, [100].log_data[83].valid := 1,
        [100].log_data[84].valid := 1, [100].log_data[85].valid := 1, [100].log_data[86].valid := 1, [100].log_data[87].valid := 1, [100].log_data[88].valid := 1, [100].log_data[89].valid := 1, [100].log_data[90].valid := 1, [100].log_data[91].valid := 1, [100].log_data[92].valid := 1, [100].log_data[93].valid := 1, [100].log_data[94].valid := 1, [100].log_data[95].valid := 1, [100].log_data[96].valid := 1, [100].log_data[97].valid := 1, [100].log_data[98].valid := 1, [100].log_data[99].valid := 1, [100].log_data[100].valid := 1, [100].log_data[101].valid := 1, [100].log_data[102].valid := 1, [100].log_data[103].valid := 1, [100].log_data[104].valid := 1, [100].log_data[105].valid := 1, [100].log_data[106].valid := 1, [100].log_data[107].valid := 1, [100].log_data[108].valid := 1, [100].log_data[109].valid := 1, [100].log_data[110].valid := 1, [100].log_data[111].valid := 1, [100].log_data[112].valid := 1, [100].log_data[113].valid := 1, [100].log_data[114].valid := 1, [100].log_data[115].valid := 1, [100].log_data[116].valid := 1, [100].log_data[117].valid := 1, [100].log_data[118].valid := 1, [100].log_data[119].valid := 1, [100].log_data[120].valid := 1, [100].log_data[121].valid := 1, [100].log_data[122].valid := 1, [100].log_data[123].valid := 1, [100].log_data[124].valid := 1, [100].time.Year := 2023, [100].time.Month := 1, [100].time.Day := 17, [100].time.Hour := 7, [100].time.Minute := 59, [100].time.Second := 59, [101].log_data[0].min := 1.0, [101].log_data[0].max := 1.0, [101].log_data[0].total := 3600.0, [101].log_data[0].time := 3600.0, [101].log_data[0].valid := 1, [101].log_data[1].time := 3600.0, [101].log_data[1].valid := 1, [101].log_data[2].time := 3600.0, [101].log_data[2].valid := 1, [101].log_data[3].time := 3600.0, [101].log_data[3].valid := 1, [101].log_data[4].time := 3600.0, [101].log_data[4].valid := 1,
        [101].log_data[5].time := 3600.0, [101].log_data[5].valid := 1, [101].log_data[6].time := 3600.0, [101].log_data[6].valid := 1, [101].log_data[7].time := 3600.0, [101].log_data[7].valid := 1, [101].log_data[8].max := 1.0, [101].log_data[8].total := 1475.0, [101].log_data[8].time := 3600.0, [101].log_data[8].minminute := 14, [101].log_data[8].valid := 1, [101].log_data[9].max := 1.0, [101].log_data[9].total := 1466.251, [101].log_data[9].time := 3600.0, [101].log_data[9].minminute := 14, [101].log_data[9].valid := 1, [101].log_data[10].min := 1.0, [101].log_data[10].max := 1.0, [101].log_data[10].total := 3600.0, [101].log_data[10].time := 3600.0, [101].log_data[10].valid := 1, [101].log_data[11].time := 3600.0, [101].log_data[11].valid := 1, [101].log_data[12].min := 1.0, [101].log_data[12].max := 1.0, [101].log_data[12].total := 3600.0, [101].log_data[12].time := 3600.0, [101].log_data[12].valid := 1, [101].log_data[13].min := 1.0, [101].log_data[13].max := 1.0, [101].log_data[13].total := 3600.0, [101].log_data[13].time := 3600.0, [101].log_data[13].valid := 1, [101].log_data[14].time := 3600.0, [101].log_data[14].valid := 1, [101].log_data[15].time := 3600.0, [101].log_data[15].valid := 1, [101].log_data[16].time := 3600.0, [101].log_data[16].valid := 1, [101].log_data[17].min := 1.0, [101].log_data[17].max := 1.0, [101].log_data[17].total := 3600.0, [101].log_data[17].time := 3600.0, [101].log_data[17].valid := 1, [101].log_data[18].time := 3600.0, [101].log_data[18].valid := 1, [101].log_data[19].time := 3600.0, [101].log_data[19].valid := 1, [101].log_data[20].time := 3600.0, [101].log_data[20].valid := 1, [101].log_data[21].min := 1.0, [101].log_data[21].max := 1.0, [101].log_data[21].total := 3600.0, [101].log_data[21].time := 3600.0, [101].log_data[21].valid := 1, [101].log_data[22].time := 3600.0, [101].log_data[22].valid := 1, [101].log_data[23].time := 3600.0, [101].log_data[23].valid := 1, [101].log_data[24].time := 3600.0,
        [101].log_data[24].valid := 1, [101].log_data[25].time := 3600.0, [101].log_data[25].valid := 1, [101].log_data[26].time := 3600.0, [101].log_data[26].valid := 1, [101].log_data[27].time := 3600.0, [101].log_data[27].valid := 1, [101].log_data[28].time := 3600.0, [101].log_data[28].valid := 1, [101].log_data[29].min := 1.0, [101].log_data[29].max := 1.0, [101].log_data[29].total := 3600.0, [101].log_data[29].time := 3600.0, [101].log_data[29].valid := 1, [101].log_data[30].min := 1.0, [101].log_data[30].max := 1.0, [101].log_data[30].total := 3600.0, [101].log_data[30].time := 3600.0, [101].log_data[30].valid := 1, [101].log_data[31].max := 1.0, [101].log_data[31].total := 770.0, [101].log_data[31].time := 3600.0, [101].log_data[31].minminute := 3, [101].log_data[31].valid := 1, [101].log_data[32].max := 1.0, [101].log_data[32].total := 543.249, [101].log_data[32].time := 3600.0, [101].log_data[32].maxminute := 5, [101].log_data[32].valid := 1, [101].log_data[33].time := 3600.0, [101].log_data[33].valid := 1, [101].log_data[34].time := 3600.0, [101].log_data[34].valid := 1, [101].log_data[35].max := 1.0, [101].log_data[35].total := 731.99805, [101].log_data[35].time := 3600.0, [101].log_data[35].minminute := 8, [101].log_data[35].valid := 1, [101].log_data[36].max := 1.0, [101].log_data[36].total := 511.24698, [101].log_data[36].time := 3600.0, [101].log_data[36].maxminute := 9, [101].log_data[36].valid := 1, [101].log_data[37].time := 3600.0, [101].log_data[37].valid := 1, [101].log_data[38].time := 3600.0, [101].log_data[38].valid := 1, [101].log_data[39].min := 0.9956484, [101].log_data[39].max := 1.005306, [101].log_data[39].total := 3604.653, [101].log_data[39].time := 3600.0, [101].log_data[39].minminute := 26, [101].log_data[39].maxminute := 10, [101].log_data[39].valid := 1, [101].log_data[40].min := 7.5942707, [101].log_data[40].max := 7.604989, [101].log_data[40].total := 27362.275, [101].log_data[40].time := 3600.0, [101].log_data[40].minminute := 27, [101].log_data[40].maxminute := 44,
        [101].log_data[40].valid := 1, [101].log_data[41].min := 0.02273633, [101].log_data[41].max := 0.023128908, [101].log_data[41].total := 82.52552, [101].log_data[41].time := 3600.0, [101].log_data[41].valid := 1, [101].log_data[42].min := 2.2916427, [101].log_data[42].max := 2.2960005, [101].log_data[42].total := 8258.851, [101].log_data[42].time := 3600.0, [101].log_data[42].minminute := 13, [101].log_data[42].maxminute := 11, [101].log_data[42].valid := 1, [101].log_data[43].min := -0.27999878, [101].log_data[43].max := -0.26000214, [101].log_data[43].total := -962.73615, [101].log_data[43].time := 3600.0, [101].log_data[43].maxminute := 4, [101].log_data[43].valid := 1, [101].log_data[44].min := -0.3199997, [101].log_data[44].max := -0.27999878, [101].log_data[44].total := -1068.9395, [101].log_data[44].time := 3600.0, [101].log_data[44].maxminute := 24, [101].log_data[44].valid := 1, [101].log_data[45].time := 3600.0, [101].log_data[45].valid := 1, [101].log_data[46].time := 3600.0, [101].log_data[46].valid := 1, [101].log_data[47].time := 3600.0, [101].log_data[47].valid := 1, [101].log_data[48].min := 6.739343, [101].log_data[48].max := 6.752809, [101].log_data[48].total := 24278.322, [101].log_data[48].time := 3600.0, [101].log_data[48].minminute := 18, [101].log_data[48].maxminute := 59, [101].log_data[48].valid := 1, [101].log_data[49].min := 9.465334, [101].log_data[49].max := 9.551309, [101].log_data[49].total := 34260.145, [101].log_data[49].time := 3600.0, [101].log_data[49].maxminute := 54, [101].log_data[49].valid := 1, [101].log_data[50].min := 1.9728262, [101].log_data[50].max := 2.1063828, [101].log_data[50].total := 7414.7524, [101].log_data[50].time := 3600.0, [101].log_data[50].minminute := 59, [101].log_data[50].maxminute := 47, [101].log_data[50].valid := 1, [101].log_data[51].time := 3600.0, [101].log_data[51].valid := 1, [101].log_data[52].min := -4.5599976, [101].log_data[52].max := 0.11999512, [101].log_data[52].total := -6250.8276, [101].log_data[52].time := 3600.0, [101].log_data[52].minminute := 50, [101].log_data[52].maxminute := 3, [101].log_data[52].valid := 1,
        [101].log_data[53].min := -4.2599945, [101].log_data[53].max := 0.2400055, [101].log_data[53].total := -5697.344, [101].log_data[53].time := 3600.0, [101].log_data[53].minminute := 50, [101].log_data[53].maxminute := 9, [101].log_data[53].valid := 1, [101].log_data[54].max := 0.5375, [101].log_data[54].total := 519.72144, [101].log_data[54].time := 3600.0, [101].log_data[54].minminute := 3, [101].log_data[54].maxminute := 50, [101].log_data[54].valid := 1, [101].log_data[55].max := 0.568, [101].log_data[55].total := 488.6963, [101].log_data[55].time := 3600.0, [101].log_data[55].minminute := 8, [101].log_data[55].maxminute := 50, [101].log_data[55].valid := 1, [101].log_data[56].min := 0.15965673, [101].log_data[56].max := 0.16020635, [101].log_data[56].total := 575.5848, [101].log_data[56].time := 3600.0, [101].log_data[56].maxminute := 44, [101].log_data[56].valid := 1, [101].log_data[57].min := 0.23440449, [101].log_data[57].max := 0.23507187, [101].log_data[57].total := 844.5412, [101].log_data[57].time := 3600.0, [101].log_data[57].minminute := 1, [101].log_data[57].maxminute := 30, [101].log_data[57].valid := 1, [101].log_data[58].time := 3600.0, [101].log_data[58].valid := 1, [101].log_data[59].time := 3600.0, [101].log_data[59].valid := 1, [101].log_data[60].valid := 1, [101].log_data[61].valid := 1, [101].log_data[62].valid := 1, [101].log_data[63].valid := 1, [101].log_data[64].valid := 1, [101].log_data[65].valid := 1, [101].log_data[66].valid := 1, [101].log_data[67].valid := 1, [101].log_data[68].valid := 1, [101].log_data[69].valid := 1, [101].log_data[70].valid := 1, [101].log_data[71].valid := 1, [101].log_data[72].valid := 1, [101].log_data[73].valid := 1, [101].log_data[74].valid := 1, [101].log_data[75].valid := 1, [101].log_data[76].valid := 1, [101].log_data[77].valid := 1, [101].log_data[78].valid := 1, [101].log_data[79].valid := 1, [101].log_data[80].valid := 1, [101].log_data[81].valid := 1, [101].log_data[82].valid := 1, [101].log_data[83].valid := 1,
        [101].log_data[84].valid := 1, [101].log_data[85].valid := 1, [101].log_data[86].valid := 1, [101].log_data[87].valid := 1, [101].log_data[88].valid := 1, [101].log_data[89].valid := 1, [101].log_data[90].valid := 1, [101].log_data[91].valid := 1, [101].log_data[92].valid := 1, [101].log_data[93].valid := 1, [101].log_data[94].valid := 1, [101].log_data[95].valid := 1, [101].log_data[96].valid := 1, [101].log_data[97].valid := 1, [101].log_data[98].valid := 1, [101].log_data[99].valid := 1, [101].log_data[100].valid := 1, [101].log_data[101].valid := 1, [101].log_data[102].valid := 1, [101].log_data[103].valid := 1, [101].log_data[104].valid := 1, [101].log_data[105].valid := 1, [101].log_data[106].valid := 1, [101].log_data[107].valid := 1, [101].log_data[108].valid := 1, [101].log_data[109].valid := 1, [101].log_data[110].valid := 1, [101].log_data[111].valid := 1, [101].log_data[112].valid := 1, [101].log_data[113].valid := 1, [101].log_data[114].valid := 1, [101].log_data[115].valid := 1, [101].log_data[116].valid := 1, [101].log_data[117].valid := 1, [101].log_data[118].valid := 1, [101].log_data[119].valid := 1, [101].log_data[120].valid := 1, [101].log_data[121].valid := 1, [101].log_data[122].valid := 1, [101].log_data[123].valid := 1, [101].log_data[124].valid := 1, [101].time.Year := 2023, [101].time.Month := 1, [101].time.Day := 17, [101].time.Hour := 8, [101].time.Minute := 59, [101].time.Second := 59, [102].log_data[0].min := 1.0, [102].log_data[0].max := 1.0, [102].log_data[0].total := 3599.5, [102].log_data[0].time := 3599.5, [102].log_data[0].valid := 1, [102].log_data[1].max := 1.0, [102].log_data[1].total := 535.5, [102].log_data[1].time := 3599.5, [102].log_data[1].maxminute := 17, [102].log_data[1].valid := 1, [102].log_data[2].max := 1.0, [102].log_data[2].total := 532.0, [102].log_data[2].time := 3599.5,
        [102].log_data[2].maxminute := 17, [102].log_data[2].valid := 1, [102].log_data[3].time := 3599.5, [102].log_data[3].valid := 1, [102].log_data[4].time := 3599.5, [102].log_data[4].valid := 1, [102].log_data[5].max := 1.0, [102].log_data[5].total := 240.0, [102].log_data[5].time := 3599.5, [102].log_data[5].maxminute := 20, [102].log_data[5].valid := 1, [102].log_data[6].time := 3599.5, [102].log_data[6].valid := 1, [102].log_data[7].time := 3599.5, [102].log_data[7].valid := 1, [102].log_data[8].min := 1.0, [102].log_data[8].max := 1.0, [102].log_data[8].total := 3599.5, [102].log_data[8].time := 3599.5, [102].log_data[8].valid := 1, [102].log_data[9].min := 1.0, [102].log_data[9].max := 1.0, [102].log_data[9].total := 3599.5, [102].log_data[9].time := 3599.5, [102].log_data[9].valid := 1, [102].log_data[10].min := 1.0, [102].log_data[10].max := 1.0, [102].log_data[10].total := 3599.5, [102].log_data[10].time := 3599.5, [102].log_data[10].valid := 1, [102].log_data[11].time := 3599.5, [102].log_data[11].valid := 1, [102].log_data[12].min := 1.0, [102].log_data[12].max := 1.0, [102].log_data[12].total := 3599.5, [102].log_data[12].time := 3599.5, [102].log_data[12].valid := 1, [102].log_data[13].min := 1.0, [102].log_data[13].max := 1.0, [102].log_data[13].total := 3599.5, [102].log_data[13].time := 3599.5, [102].log_data[13].valid := 1, [102].log_data[14].time := 3599.5, [102].log_data[14].valid := 1, [102].log_data[15].time := 3599.5, [102].log_data[15].valid := 1, [102].log_data[16].time := 3599.5, [102].log_data[16].valid := 1, [102].log_data[17].min := 1.0, [102].log_data[17].max := 1.0, [102].log_data[17].total := 3599.5, [102].log_data[17].time := 3599.5, [102].log_data[17].valid := 1, [102].log_data[18].time := 3599.5, [102].log_data[18].valid := 1, [102].log_data[19].time := 3599.5, [102].log_data[19].valid := 1, [102].log_data[20].time := 3599.5, [102].log_data[20].valid := 1, [102].log_data[21].min := 1.0,
        [102].log_data[21].max := 1.0, [102].log_data[21].total := 3599.5, [102].log_data[21].time := 3599.5, [102].log_data[21].valid := 1, [102].log_data[22].time := 3599.5, [102].log_data[22].valid := 1, [102].log_data[23].time := 3599.5, [102].log_data[23].valid := 1, [102].log_data[24].time := 3599.5, [102].log_data[24].valid := 1, [102].log_data[25].time := 3599.5, [102].log_data[25].valid := 1, [102].log_data[26].time := 3599.5, [102].log_data[26].valid := 1, [102].log_data[27].time := 3599.5, [102].log_data[27].valid := 1, [102].log_data[28].time := 3599.5, [102].log_data[28].valid := 1, [102].log_data[29].min := 1.0, [102].log_data[29].max := 1.0, [102].log_data[29].total := 3599.5, [102].log_data[29].time := 3599.5, [102].log_data[29].valid := 1, [102].log_data[30].min := 1.0, [102].log_data[30].max := 1.0, [102].log_data[30].total := 3599.5, [102].log_data[30].time := 3599.5, [102].log_data[30].valid := 1, [102].log_data[31].max := 1.0, [102].log_data[31].total := 1440.2471, [102].log_data[31].time := 3599.5, [102].log_data[31].valid := 1, [102].log_data[32].max := 1.0, [102].log_data[32].total := 1629.7471, [102].log_data[32].time := 3599.5, [102].log_data[32].maxminute := 1, [102].log_data[32].valid := 1, [102].log_data[33].time := 3599.5, [102].log_data[33].valid := 1, [102].log_data[34].time := 3599.5, [102].log_data[34].valid := 1, [102].log_data[35].max := 1.0, [102].log_data[35].total := 1629.7471, [102].log_data[35].time := 3599.5, [102].log_data[35].maxminute := 7, [102].log_data[35].valid := 1, [102].log_data[36].max := 1.0, [102].log_data[36].total := 1440.2471, [102].log_data[36].time := 3599.5, [102].log_data[36].minminute := 5, [102].log_data[36].valid := 1, [102].log_data[37].max := 7.578744, [102].log_data[37].total := 3517.7424, [102].log_data[37].time := 3599.5, [102].log_data[37].maxminute := 18, [102].log_data[37].valid := 1, [102].log_data[38].time := 3599.5, [102].log_data[38].valid := 1, [102].log_data[39].min := 0.994824, [102].log_data[39].max := 1.0215589,
        [102].log_data[39].total := 3607.4558, [102].log_data[39].time := 3599.5, [102].log_data[39].minminute := 45, [102].log_data[39].maxminute := 20, [102].log_data[39].valid := 1, [102].log_data[40].min := 7.584652, [102].log_data[40].max := 7.6104846, [102].log_data[40].total := 27360.346, [102].log_data[40].time := 3599.5, [102].log_data[40].minminute := 39, [102].log_data[40].maxminute := 41, [102].log_data[40].valid := 1, [102].log_data[41].min := 0.022540038, [102].log_data[41].max := 0.02411035, [102].log_data[41].total := 82.44948, [102].log_data[41].time := 3599.5, [102].log_data[41].minminute := 29, [102].log_data[41].maxminute := 55, [102].log_data[41].valid := 1, [102].log_data[42].min := 2.2910538, [102].log_data[42].max := 2.2963536, [102].log_data[42].total := 8257.591, [102].log_data[42].time := 3599.5, [102].log_data[42].minminute := 6, [102].log_data[42].maxminute := 47, [102].log_data[42].valid := 1, [102].log_data[43].min := -0.27999878, [102].log_data[43].max := -0.26000214, [102].log_data[43].total := -959.9876, [102].log_data[43].time := 3599.5, [102].log_data[43].minminute := 4, [102].log_data[43].valid := 1, [102].log_data[44].min := -0.3199997, [102].log_data[44].max := -0.30000305, [102].log_data[44].total := -1079.9661, [102].log_data[44].time := 3599.5, [102].log_data[44].minminute := 44, [102].log_data[44].valid := 1, [102].log_data[45].time := 3599.5, [102].log_data[45].valid := 1, [102].log_data[46].time := 3599.5, [102].log_data[46].valid := 1, [102].log_data[47].time := 3599.5, [102].log_data[47].valid := 1, [102].log_data[48].min := 6.5681376, [102].log_data[48].max := 6.9534187, [102].log_data[48].total := 24174.88, [102].log_data[48].time := 3599.5, [102].log_data[48].minminute := 47, [102].log_data[48].maxminute := 23, [102].log_data[48].valid := 1, [102].log_data[49].min := 6.8048, [102].log_data[49].max := 9.534036, [102].log_data[49].total := 29686.87, [102].log_data[49].time := 3599.5, [102].log_data[49].minminute := 49, [102].log_data[49].maxminute := 14, [102].log_data[49].valid := 1, [102].log_data[50].min := 1.9466803, [102].log_data[50].max := 2.060804,
        [102].log_data[50].total := 7236.2856, [102].log_data[50].time := 3599.5, [102].log_data[50].minminute := 19, [102].log_data[50].maxminute := 27, [102].log_data[50].valid := 1, [102].log_data[51].time := 3599.5, [102].log_data[51].valid := 1, [102].log_data[52].min := -2.9800034, [102].log_data[52].max := 0.11999512, [102].log_data[52].total := -7539.307, [102].log_data[52].time := 3599.5, [102].log_data[52].minminute := 12, [102].log_data[52].valid := 1, [102].log_data[53].min := -2.4800034, [102].log_data[53].max := 0.2599945, [102].log_data[53].total := -6945.793, [102].log_data[53].time := 3599.5, [102].log_data[53].minminute := 7, [102].log_data[53].maxminute := 49, [102].log_data[53].valid := 1, [102].log_data[54].max := 0.531, [102].log_data[54].total := 1216.9149, [102].log_data[54].time := 3599.5, [102].log_data[54].maxminute := 54, [102].log_data[54].valid := 1, [102].log_data[55].max := 0.547, [102].log_data[55].total := 1217.3497, [102].log_data[55].time := 3599.5, [102].log_data[55].minminute := 5, [102].log_data[55].maxminute := 59, [102].log_data[55].valid := 1, [102].log_data[56].min := 0.15961748, [102].log_data[56].max := 0.16012783, [102].log_data[56].total := 575.42786, [102].log_data[56].time := 3599.5, [102].log_data[56].minminute := 55, [102].log_data[56].maxminute := 7, [102].log_data[56].valid := 1, [102].log_data[57].min := 0.23240234, [102].log_data[57].max := 0.23487559, [102].log_data[57].total := 843.3228, [102].log_data[57].time := 3599.5, [102].log_data[57].minminute := 56, [102].log_data[57].maxminute := 2, [102].log_data[57].valid := 1, [102].log_data[58].time := 3599.5, [102].log_data[58].valid := 1, [102].log_data[59].time := 3599.5, [102].log_data[59].valid := 1, [102].log_data[60].valid := 1, [102].log_data[61].valid := 1, [102].log_data[62].valid := 1, [102].log_data[63].valid := 1, [102].log_data[64].valid := 1, [102].log_data[65].valid := 1, [102].log_data[66].valid := 1, [102].log_data[67].valid := 1, [102].log_data[68].valid := 1, [102].log_data[69].valid := 1, [102].log_data[70].valid := 1,
